# B&R Automation Studio project PLC code - cp (part 16)

#### AsignDataP5.st
```iecst
ACTION AsignDataP5:

	//Just writing the fixed configuration once per each 5s
	IF NOT (EDGEPOS(gPLC.xBlk_5s) OR gPLC.xFirst_Scan OR xChangedSimMachine) THEN
		RETURN;
	END_IF

	////////////////////////////////////////////////////////////
	/////GENERAL	GENERAL		GENERAL		GENERAL	////////////
	////////////////////////////////////////////////////////////

	gMachine.Pt.xControlledRemotely := FALSE;

	gMachine.Pt.CT.rMountedMediaLevelInBypassMode		:= 120.0;
	gMachine.Pt.CT.rMaxTicknessMedia		:= 120.0;
	gMachine.Pt.CT.rMinTicknessMedia		:= 2.0;
	gMachine.Pt.CT.iNumSAIInstalled			:= 2;

	gMachine.Pt.rMaxPrintHeadPos			:= 1668.0;
	gMachine.Pt.rMinPrintHeadPos			:= 10;
	gMachine.Pt.CT.rMinMarginPrinting		:= 1.0;

	gMachine.Pt.iMediaFilter 				:= 0;

	gMachine.Pt.PDSignalTpe 				:= PDCFG_SENSOR_AND_CARRIAGE;
	gMachine.Pt.xProtectPHWithStoppedMediaBended:= TRUE;
	gMachine.Pt.xProtectPHForBlowersRunning		:= FALSE;
	gMachine.Pt.Clean.xCleanBeltTopInstall 		:= FALSE;
	gMachine.Pt.xAllowLaboratory	 			:= TRUE;
	gMachine.Pt.xAllowJamRecovery	 			:= FALSE;
	gMachine.Pt.xJobNotReadyIsCritical	 		:= FALSE;
	gMachine.Pt.Clean.xCleanBeltForUv			:= FALSE;
	gMachine.Pt.CommsType						:= Type_ModbusTcp;

	gMachine.Pt.Hw.iWidth					:= 1440;
	gMachine.Pt.Hw.rMinPrintPosition		:= 2.0;
	gMachine.Pt.Hw.iMaxCuringLedBars		:= 0;
	gMachine.Pt.Hw.xDoubleLineAllowed		:= TRUE;
	gMachine.Pt.Hw.xSuctionModeAllowed		:= FALSE;

	gMachine.St.HwData.xIsPlatform5			:= TRUE;
	gMachine.St.HwData.xIsWater				:= gMachine.Pt.MachineModel=Type_P5_WTR;
	gMachine.St.HwData.xIsCubik				:= FALSE;

	//Belt
	gBelt.parameters.xRemoteAcceleration := FALSE;
	gBelt.parameters.xRemoteDeceleration := FALSE;
	gBelt.parameters.rAcceleration := 1050;
	gBelt.parameters.rDeceleration := 1050;
	gBelt.parameters.rMaxAcceleration := 1500.0;
	gBelt.parameters.rMaxDeceleration := 2500.0;

	//Here are configured blocks in function of the machine direction
	//When machine is block then we need use correction as block physical 2 because PD is at the same distance than Block 1, for that is change process in function of machine 2 Blcoks or machine 1 block
	gBlock[1].parameters.iMotorAxisIndex := 2;
	gBlock[1].parameters.iMappingBlock := 1;
	gBlock[1].parameters.iIclaAxisIndex := 1;
	gBlock[1].parameters.Hw.ValvesCommsType := COMMS_POWERLINK;

	/////////////////////////////////////////////////////
	// Temperature Modules Check
	////////////////////////////////////////////////////
	IF	NOT(gInks[1].parSw.Temp.xTankHeaterEnabled OR
		gInks[2].parSw.Temp.xTankHeaterEnabled OR
		gInks[3].parSw.Temp.xTankHeaterEnabled OR
		gInks[4].parSw.Temp.xTankHeaterEnabled) THEN

		gBlock[1].parameters.Inks.xTankHeatEnabled1 := FALSE;
	ELSE
		gBlock[1].parameters.Inks.xTankHeatEnabled1 := TRUE;
	END_IF

	IF	NOT(gInks[5].parSw.Temp.xTankHeaterEnabled OR
		gInks[6].parSw.Temp.xTankHeaterEnabled OR
		gInks[7].parSw.Temp.xTankHeaterEnabled OR
		gInks[8].parSw.Temp.xTankHeaterEnabled) THEN

		gBlock[1].parameters.Inks.xTankHeatEnabled2 := FALSE;
	ELSE
		gBlock[1].parameters.Inks.xTankHeatEnabled2 := TRUE;
	END_IF

	/////////////////////////////////////////////////////
	/////BELT	BELT	BELT	BELT	BELT	BELT/////
	/////////////////////////////////////////////////////

	////////////////////////////////////////////////////////////
	/////BLOCK	BLOCK	BLOCK	BLOCK	BLOCK	BLOCK///////////
	////////////////////////////////////////////////////////////
	FOR iIndexBlock:=1 TO gMachine.Pt.CT.iNumBlocks DO

		//Position parameters (mm)
		gBlock[iIndexBlock].parameters.Motor.rSafePosition				:= 356.0;//Max heigh
		gBlock[iIndexBlock].parameters.Motor.rMinSafePosition			:= 5.0;	 //Min heigh
		gBlock[iIndexBlock].parameters.Motor.rCapPosition				:= 344.0;//CAP
		gBlock[iIndexBlock].parameters.Motor.rSafePositionCleanCarrier	:= 329.0;//Carrier out Safe
		gBlock[iIndexBlock].parameters.Motor.rDripBarsPosition			:= 279.0;//Drip
		gBlock[iIndexBlock].parameters.Motor.rCleanPosition				:= 335.0;//Clean
		gBlock[iIndexBlock].parameters.Motor.rWaterSpurtPosition		:= 342.0;//Water Spurt
		gBlock[iIndexBlock].parameters.rPrePrintingPos					:= 75.0;  //PrePrinting Position

		gBlock[iIndexBlock].parameters.Motor.rAutoSpeedMoveDown	:=15.0;
		gBlock[iIndexBlock].parameters.Motor.rAutoSpeedMoveUp	:=30.0;
		gBlock[iIndexBlock].parameters.Motor.xFastSpeedAllowed	:= FALSE;

		gBlock[iIndexBlock].parameters.Motor.DriveUnit.TransmissionType := TRANS_SCREW_PITCH;
		gBlock[iIndexBlock].parameters.Motor.DriveUnit.ScrewPitch.PulsesPerTurn := GC_UNITS_BY_REV_DRIVE;
		gBlock[iIndexBlock].parameters.Motor.DriveUnit.ScrewPitch.GearBox := 7.25;
		gBlock[iIndexBlock].parameters.Motor.DriveUnit.ScrewPitch.Pitch := 5.0;

		gBlock[iIndexBlock].parameters.Motor.rReferencePosition		:= 15.5;

		//Current Parameters
		gBlock[iIndexBlock].parameters.Motor.uiMaxCurrentBarsUp			:= 3;
		gBlock[iIndexBlock].parameters.Motor.uiMaxCurrentBarsDown		:= 1;

		gBlock[iIndexBlock].parameters.Motor.VerticalDirection:= MOTOR_POSITIVE;

		gBlock[iIndexBlock].parameters.Motor.rAcceleration		:= 172.5;
		gBlock[iIndexBlock].parameters.Motor.rDeceleration		:= 172.5;

		gBlock[iIndexBlock].parameters.Icla.DriveUnit.TransmissionType:=TRANS_LINEAL_PERIMETER;
		gBlock[iIndexBlock].parameters.Icla.DriveUnit.LinealPerimeter.GearBox:=92;
		gBlock[iIndexBlock].parameters.Icla.DriveUnit.LinealPerimeter.Perimeter:=180;
		gBlock[iIndexBlock].parameters.Icla.DriveUnit.LinealPerimeter.PulsesPerTurn:=12;

		gBlock[iIndexBlock].parameters.Inks.iMaxMachinePrintBars	:= 8;
		gBlock[iIndexBlock].parameters.Inks.iMaxBlockPrintBars		:= 8;
		gBlock[iIndexBlock].parameters.Inks.iMaxPSUwattsForBars		:= 3000;

		gBlock[iIndexBlock].parameters.xCappingProcess := FALSE;

		gBlock[iIndexBlock].parameters.Hw.SafetySignals := SAFETY_ESTOP_CALCULATED;

		//[RGP] Due to issue SUSTPLATF-236
		gBlock[iIndexBlock].parameters.xMotorOffsetAllowed := FALSE;

		gBlock[iIndexBlock].parameters.iApplicationBars := 8;
	END_FOR

	///////////////////////////////////////////////////
	/////PHOTOCELLS		PHOTOCELLS		PHOTOCELLS/////
	///////////////////////////////////////////////////

	gPhotoCells.parameters.xInstall := TRUE;
	gMachine.parSw.Hw.xInstallnSensor := FALSE;
	gPhotoCells.parameters.xSensorsPosHybridBehaviour := FALSE;

	gPhotoCells.parameters.MotorType := STP_STEPPER;
	gPhotoCells.parameters.AlignmentProcess := STP_ALIGNMENT_NO_REQUIRED;

	gPhotoCells.parameters.Speed:=2.5;
	gPhotoCells.parameters.JogSpeed:=1;
	gPhotoCells.parameters.Acceleration:=5;

	gPhotoCells.parameters.DriveUnit.TransmissionType := TRANS_SCREW_PITCH;
	gPhotoCells.parameters.DriveUnit.ScrewPitch.PulsesPerTurn := GC_UNITS_BY_REV_DRIVE;
	gPhotoCells.parameters.DriveUnit.ScrewPitch.GearBox := 1;
	gPhotoCells.parameters.DriveUnit.ScrewPitch.Pitch := 2.5;

	IF gMachine.Pt.ConfigNameID = GC_CONFIG_SIMTEST_ID THEN
		// In Simulation
		gPhotoCells.parameters.IndexDriveMaster:=4;
		gPhotoCells.parameters.IndexDriveSecondary:=5;
	ELSE
		gPhotoCells.parameters.IndexDriveMaster:=3;
		gPhotoCells.parameters.IndexDriveSecondary:=4;
	END_IF

	gPhotoCells.parameters.iSensorQuantity := 3;
	gPhotoCells.parameters.iSensorToReference := 2;
	gPhotoCells.parameters.rOffsetPosition := 0.0;
	gPhotoCells.parameters.rSensorMechPositionByPass := 60.0;//110.0; //ALX -> ToReview
	gPhotoCells.parameters.Sensors[2].rDistanceRelativeToFirstSensor := 4;
	gPhotoCells.parameters.Sensors[3].rDistanceRelativeToFirstSensor := 8;
	gPhotoCells.parameters.xEnableMountedAlrByPass := TRUE;

	//Digital Inputs
	gPhotoCells.Inputs.Signals.pInput[1] := ADR(X20DIF371_003.DInput[13]);
	gPhotoCells.Inputs.Signals.pInput[2] := ADR(X20DIF371_003.DInput[14]);
	gPhotoCells.Inputs.Signals.pInput[3] := ADR(X20DIF371_003.DInput[15]);
	gPhotoCells.Inputs.Signals.xSafetyEnable := gMachine.In.xSafetyEnabled;

	stepperMotor ACCESS ADR (gAxis[gPhotoCells.parameters.IndexDriveMaster]);
	stepperMotor.Parameter.Direction:= MOTOR_NEGATIVE_AXIS;

	///////////////////////////////////////////////////
	/////DING		DING		DING		DING  /////
	///////////////////////////////////////////////////
	gDing.Parameters.xDingInstalled := FALSE;

	/////////////////////////////////////////////////////
	/////THICKNESS		THICKNESS		 THICKNESS///////
	/////////////////////////////////////////////////////

	gThicknessCtrl.parameters.iTotalBlocksLengh := 305;
	gThicknessCtrl.parameters.Belt.iDistanceEmptyBeltIni := 455; //The difference between Long and NotLong machine is 1350mm by side [700-135=615]

	gThicknessCtrl.parameters.xMarginForBendTile := TRUE;
	gThicknessCtrl.parameters.rSafetyMarginToHeight := 3.0;

	gThicknessCtrl.parameters.sections[1].xEnabled	:= TRUE;
	gThicknessCtrl.parameters.sections[1].iStart	:= 1;
	gThicknessCtrl.parameters.sections[1].iEnd		:= 305;

	gThicknessCtrl.parameters.Detection.ProductDetect.xLoadMedia := FALSE;
	gThicknessCtrl.parameters.Detection.ProductDetect.iSensorPosition := 25;
	gThicknessCtrl.parameters.Detection.Array.xLoadMedia := TRUE;
	gThicknessCtrl.parameters.Detection.Analog.iSensorPosition := 0;
	gThicknessCtrl.parameters.Detection.Analog.xLoadMedia := TRUE;
	gThicknessCtrl.parameters.Detection.Array.iSensorPosition := 0;

	/////////////////////////////////////////////////////
	/////   TRANSPORT_VACUUM  TRANSPORT_VACUUM   ////////
	/////////////////////////////////////////////////////
	gTransVacuum[1].Parameters.xInstalled := FALSE;
	gTransVacuum[2].Parameters.xInstalled := FALSE;

	/////////////////////////////////////////////////////
	/////   NON_CRASH    NON_CRASH    NON_CRASH  ////////
	/////////////////////////////////////////////////////
	gNonCrash[1].Parameters.xInstalled := FALSE;

	/////////////////////////////////////////////////////
	/////   PLC CARDS	PLC CARDS	PLC CARDS	 ////////
	/////////////////////////////////////////////////////
	IF gPlcCards[0].Type <> CARD_UNDEFINED THEN
		RETURN;
	END_IF

	//Force "ModuleOk" in cards without it
	X20CPUData.ModuleOk := TRUE;

	AsignCardsP5;

END_ACTION

ACTION AsignCardsP5:

	gPlcCards[0].Type := CARD_CPU0484;
	gPlcCards[0].pCard := ADR(X20CPUData);
	gPlcCards[0].RequiredForFunctions[0] := CARDREQUIRED_ALWAYS;
	gPlcCards[0].stCardName := 'X20CP0483_000';
	gPlcCards[0].Location := CardInPrinter;
	iIndexPlcCar := 1;

	//CARD 01 X20DIF371
	gPlcCards[iIndexPlcCar].Type := CARD_DI16;
	gPlcCards[iIndexPlcCar].pCard := ADR(X20DIF371_001);
	gPlcCards[iIndexPlcCar].RequiredForFunctions[0] := CARDREQUIRED_ALWAYS;
	gPlcCards[iIndexPlcCar].stCardName := 'X20DIF371-001';
	gPlcCards[iIndexPlcCar].Texts[1].Details := 'Machine Config-Bit 0';
	gPlcCards[iIndexPlcCar].Texts[2].Details := 'Machine Config-Bit 1';
	gPlcCards[iIndexPlcCar].Texts[3].Details := 'Machine Config-Bit 2';
	gPlcCards[iIndexPlcCar].Texts[4].Details := 'Machine Config-Bit 3';
	gPlcCards[iIndexPlcCar].Texts[5].Details := 'Machine Config-Bit 4';
	gPlcCards[iIndexPlcCar].Texts[6].Details := 'Machine Config-Bit 5';
	gPlcCards[iIndexPlcCar].Texts[7].Details := 'Start';
	gPlcCards[iIndexPlcCar].Texts[8].Details := 'Stop';
	gPlcCards[iIndexPlcCar].Texts[9].Details := 'Automatic';
	gPlcCards[iIndexPlcCar].Texts[10].Details := 'Zero';
	gPlcCards[iIndexPlcCar].Texts[11].Details := 'Manual';
	gPlcCards[iIndexPlcCar].Texts[12].Details := 'Validation to PLC';
	gPlcCards[iIndexPlcCar].Texts[13].Details := 'CB to PLC - Print Trigger L1';
	gPlcCards[iIndexPlcCar].Texts[14].Details := 'CB to PLC - Print Trigger L2';
	gPlcCards[iIndexPlcCar].Texts[15].Details := 'Spare';
	gPlcCards[iIndexPlcCar].Texts[16].Details := 'Spare';
	gPlcCards[iIndexPlcCar].Location := CardInPrinter;
	iIndexPlcCar := iIndexPlcCar + 1;

	//CARD 02 X20DIF371
	gPlcCards[iIndexPlcCar].Type := CARD_DI16;
	gPlcCards[iIndexPlcCar].pCard := ADR(X20DIF371_002);
	gPlcCards[iIndexPlcCar].RequiredForFunctions[0] := CARDREQUIRED_ALWAYS;
	gPlcCards[iIndexPlcCar].stCardName := 'X20DIF371-002';
	gPlcCards[iIndexPlcCar].Texts[1].Details := 'Bar A-48 VDC POWER OK';
	gPlcCards[iIndexPlcCar].Texts[2].Details := 'Bar B-48 VDC POWER OK';
	gPlcCards[iIndexPlcCar].Texts[3].Details := 'Bar C-48 VDC POWER OK';
	gPlcCards[iIndexPlcCar].Texts[4].Details := 'Bar D-48 VDC POWER OK';
	gPlcCards[iIndexPlcCar].Texts[5].Details := 'Bar E-48 VDC POWER OK';
	gPlcCards[iIndexPlcCar].Texts[6].Details := 'Bar F-48 VDC POWER OK';
	gPlcCards[iIndexPlcCar].Texts[7].Details := 'Bar G-48 VDC POWER OK';
	gPlcCards[iIndexPlcCar].Texts[8].Details := 'Bar H-48 VDC POWER OK';
	gPlcCards[iIndexPlcCar].Texts[9].Details := 'Bars heater - 48 VDC POWER OK';
	gPlcCards[iIndexPlcCar].Texts[10].Details := 'Transp driver-Diff contact alarm';
	gPlcCards[iIndexPlcCar].Texts[11].Details := 'Elev. driver-CB contact alarm';
	gPlcCards[iIndexPlcCar].Texts[12].Details := '48 VDC PSUs-Diff contact alarm';
	gPlcCards[iIndexPlcCar].Texts[13].Details := '24 VDC PSUs-IDS power alarm';
	gPlcCards[iIndexPlcCar].Texts[14].Details := 'Front light curtain-Alarm';
	gPlcCards[iIndexPlcCar].Texts[15].Details := 'Back Safety Switch-Alarm';
	gPlcCards[iIndexPlcCar].Texts[16].Details := 'Safety module status-Safety OK';
	gPlcCards[iIndexPlcCar].Location := CardInPrinter;
	iIndexPlcCar := iIndexPlcCar + 1;

	//CARD 03 X20DIF371
	gPlcCards[iIndexPlcCar].Type := CARD_DI16;
	gPlcCards[iIndexPlcCar].pCard := ADR(X20DIF371_003);
	gPlcCards[iIndexPlcCar].RequiredForFunctions[0] := CARDREQUIRED_ALWAYS;
	gPlcCards[iIndexPlcCar].stCardName := 'X20DIF371-003';
	gPlcCards[iIndexPlcCar].Texts[1].Details := 'UPS 1 - Failure UPS';
	gPlcCards[iIndexPlcCar].Texts[2].Details := 'UPS 1 - Utility Failure';
	gPlcCards[iIndexPlcCar].Texts[3].Details := 'UPS 1 - Low Battery';
	gPlcCards[iIndexPlcCar].Texts[4].Details := 'UPS 1 - Inverter Failure';
	gPlcCards[iIndexPlcCar].Texts[5].Details := 'UPS 2 - Failure UPS';
	gPlcCards[iIndexPlcCar].Texts[6].Details := 'UPS 2 - Utility Failure';
	gPlcCards[iIndexPlcCar].Texts[7].Details := 'UPS 2 - Low Battery';
	gPlcCards[iIndexPlcCar].Texts[8].Details := 'UPS 2 - Inverter Failure';
	gPlcCards[iIndexPlcCar].Texts[9].Details := 'Bars ref. sensor - ON signal';
	gPlcCards[iIndexPlcCar].Texts[10].Details := 'Spare';
	gPlcCards[iIndexPlcCar].Texts[11].Details := 'PD - Broken sensor alarm';
	gPlcCards[iIndexPlcCar].Texts[12].Details := 'DPT - Broken sensor alarm';
	gPlcCards[iIndexPlcCar].Texts[13].Details := '3L - Detected tile (Photocell 1)';
	gPlcCards[iIndexPlcCar].Texts[14].Details := '3L - Bent tile (Photocell 2)';
	gPlcCards[iIndexPlcCar].Texts[15].Details := '3L - Mounted tile (Photocell 3)';
	gPlcCards[iIndexPlcCar].Texts[16].Details := 'Spare';
	gPlcCards[iIndexPlcCar].Location := CardInPrinter;
	iIndexPlcCar := iIndexPlcCar + 1;

	//CARD 04 X20DIF371
	gPlcCards[iIndexPlcCar].Type := CARD_DI16;
	gPlcCards[iIndexPlcCar].pCard := ADR(X20DIF371_004);
	gPlcCards[iIndexPlcCar].RequiredForFunctions[0] := CARDREQUIRED_ALWAYS;
	gPlcCards[iIndexPlcCar].stCardName := 'X20DIF371-004';
	gPlcCards[iIndexPlcCar].Texts[1].Details := 'Bar A - Klixon';
	gPlcCards[iIndexPlcCar].Texts[2].Details := 'Bar B - Klixon';
	gPlcCards[iIndexPlcCar].Texts[3].Details := 'Bar C - Klixon';
	gPlcCards[iIndexPlcCar].Texts[4].Details := 'Bar D - Klixon';
	gPlcCards[iIndexPlcCar].Texts[5].Details := 'Bar E - Klixon';
	gPlcCards[iIndexPlcCar].Texts[6].Details := 'Bar F - Klixon';
	gPlcCards[iIndexPlcCar].Texts[7].Details := 'Bar G - Klixon';
	gPlcCards[iIndexPlcCar].Texts[8].Details := 'Bar H - Klixon';
	gPlcCards[iIndexPlcCar].Texts[9].Details := 'Tank A - Empty Level';
	gPlcCards[iIndexPlcCar].Texts[10].Details := 'Tank B - Empty Level';
	gPlcCards[iIndexPlcCar].Texts[11].Details := 'Tank C - Empty Level';
	gPlcCards[iIndexPlcCar].Texts[12].Details := 'Tank D - Empty Level';
	gPlcCards[iIndexPlcCar].Texts[13].Details := 'Tank E - Empty Level';
	gPlcCards[iIndexPlcCar].Texts[14].Details := 'Tank F - Empty Level';
	gPlcCards[iIndexPlcCar].Texts[15].Details := 'Tank G - Empty Level';
	gPlcCards[iIndexPlcCar].Texts[16].Details := 'Tank H - Empty Level';
	gPlcCards[iIndexPlcCar].Location := CardInPrinter;
	iIndexPlcCar := iIndexPlcCar + 1;

	//CARD 05 X20DIF371
	gPlcCards[iIndexPlcCar].Type := CARD_DI16;
	gPlcCards[iIndexPlcCar].pCard := ADR(X20DIF371_005);
	gPlcCards[iIndexPlcCar].RequiredForFunctions[0] := CARDREQUIRED_ALWAYS;
	gPlcCards[iIndexPlcCar].stCardName := 'X20DIF371-005';
	gPlcCards[iIndexPlcCar].Texts[1].Details := 'Tank A - Full Level';
	gPlcCards[iIndexPlcCar].Texts[2].Details := 'Tank B - Full Level';
	gPlcCards[iIndexPlcCar].Texts[3].Details := 'Tank C - Full Level';
	gPlcCards[iIndexPlcCar].Texts[4].Details := 'Tank D - Full Level';
	gPlcCards[iIndexPlcCar].Texts[5].Details := 'Tank E - Full Level';
	gPlcCards[iIndexPlcCar].Texts[6].Details := 'Tank F - Full Level';
	gPlcCards[iIndexPlcCar].Texts[7].Details := 'Tank G - Full Level';
	gPlcCards[iIndexPlcCar].Texts[8].Details := 'Tank H - Full Level';
	gPlcCards[iIndexPlcCar].Texts[9].Details := 'Tank A - Pressure Switch';
	gPlcCards[iIndexPlcCar].Texts[10].Details := 'Tank B - Pressure Switch';
	gPlcCards[iIndexPlcCar].Texts[11].Details := 'Tank C - Pressure Switch';
	gPlcCards[iIndexPlcCar].Texts[12].Details := 'Tank D - Pressure Switch';
	gPlcCards[iIndexPlcCar].Texts[13].Details := 'Tank E - Pressure Switch';
	gPlcCards[iIndexPlcCar].Texts[14].Details := 'Tank F - Pressure Switch';
	gPlcCards[iIndexPlcCar].Texts[15].Details := 'Tank G - Pressure Switch';
	gPlcCards[iIndexPlcCar].Texts[16].Details := 'Tank H - Pressure Switch';
	gPlcCards[iIndexPlcCar].Location := CardInPrinter;
	iIndexPlcCar := iIndexPlcCar + 1;

	//CARD 06 X20DIF371
	gPlcCards[iIndexPlcCar].Type := CARD_DI16;
	gPlcCards[iIndexPlcCar].pCard := ADR(X20DIF371_006);
	gPlcCards[iIndexPlcCar].RequiredForFunctions[0] := CARDREQUIRED_ALWAYS;
	gPlcCards[iIndexPlcCar].stCardName := 'X20DIF371-006';
	gPlcCards[iIndexPlcCar].Texts[1].Details := 'PBF - Bit 0';
	gPlcCards[iIndexPlcCar].Texts[2].Details := 'PBF - Bit 1';
	gPlcCards[iIndexPlcCar].Texts[3].Details := 'PBF - Bit 2';
	gPlcCards[iIndexPlcCar].Texts[4].Details := 'PBF - Bit 3';
	gPlcCards[iIndexPlcCar].Texts[5].Details := 'PBF - Bit 4';
	gPlcCards[iIndexPlcCar].Texts[6].Details := 'PBF - Bit 5';
	gPlcCards[iIndexPlcCar].Texts[7].Details := 'PBF - Bit 6';
	gPlcCards[iIndexPlcCar].Texts[8].Details := 'PBF - Bit 7';
	gPlcCards[iIndexPlcCar].Texts[9].Details := 'PBF - Strobe';
	gPlcCards[iIndexPlcCar].Texts[10].Details := 'Consent Line-Machine 1';
	gPlcCards[iIndexPlcCar].Texts[11].Details := 'Consent Line-Machine 2';
	gPlcCards[iIndexPlcCar].Texts[12].Details := 'PH External Cleaning';
	gPlcCards[iIndexPlcCar].Texts[13].Details := 'RESERVED';
	gPlcCards[iIndexPlcCar].Texts[14].Details := 'RESERVED';
	gPlcCards[iIndexPlcCar].Texts[15].Details := 'Spare';
	gPlcCards[iIndexPlcCar].Texts[16].Details := 'Spare';
	gPlcCards[iIndexPlcCar].Location := CardInPrinter;
	iIndexPlcCar := iIndexPlcCar + 1;

	//CARD 07 PS
	gPlcCards[iIndexPlcCar].Type := CARD_PS33;
	gPlcCards[iIndexPlcCar].pCard := ADR(X20PS3300_007);
	gPlcCards[iIndexPlcCar].RequiredForFunctions[0] := CARDREQUIRED_ALWAYS;
	gPlcCards[iIndexPlcCar].stCardName := 'X20PS3300-007';
	gPlcCards[iIndexPlcCar].Location := CardInPrinter;
	iIndexPlcCar := iIndexPlcCar + 1;

	//CARD 8 X20DI9372
	gPlcCards[iIndexPlcCar].Type := CARD_DI16;
	gPlcCards[iIndexPlcCar].pCard := ADR(X20DI9372_008);
	gPlcCards[iIndexPlcCar].RequiredForFunctions[0] := CARDREQUIRED_ALWAYS;
	gPlcCards[iIndexPlcCar].stCardName := 'X20DI9372_008';
	gPlcCards[iIndexPlcCar].Texts[1].Details :='48VDC PSU 1 (PH) -48 V OK';
	gPlcCards[iIndexPlcCar].Texts[2].Details :='48VDC PSU 2 (PH) -48 V OK';
	gPlcCards[iIndexPlcCar].Texts[3].Details :='48VDC PSU 3 (PH) -48 V OK';
	gPlcCards[iIndexPlcCar].Texts[4].Details :='48VDC PSU 4 (PH) -48 V OK';
	gPlcCards[iIndexPlcCar].Texts[5].Details :='48VDC PSU 5 (PH) -48 V OK';
	gPlcCards[iIndexPlcCar].Texts[6].Details :='48VDC PSU 6 (PH) -48 V OK';
	gPlcCards[iIndexPlcCar].Texts[7].Details :='48VDC PSU 7 (Heat) -48 V OK';
	gPlcCards[iIndexPlcCar].Texts[8].Details :='48VDC PSU 8 (Heat) -48 V OK';
	gPlcCards[iIndexPlcCar].Texts[9].Details :='48VDC PSU 9 (Heat) -48 V OK';
	gPlcCards[iIndexPlcCar].Texts[10].Details :='Spare';
	gPlcCards[iIndexPlcCar].Texts[11].Details :='Spare';
	gPlcCards[iIndexPlcCar].Texts[12].Details :='Spare';
	gPlcCards[iIndexPlcCar].Location := CardInPrinter;
	iIndexPlcCar := iIndexPlcCar + 1;

	//CARD 9 X20DOF322
	gPlcCards[iIndexPlcCar].Type := CARD_DO16;
	gPlcCards[iIndexPlcCar].pCard := ADR(X20DOF322_009);
	gPlcCards[iIndexPlcCar].RequiredForFunctions[0] := CARDREQUIRED_ALWAYS;
	gPlcCards[iIndexPlcCar].stCardName := 'X20DOF322_009';
	gPlcCards[iIndexPlcCar].Texts[1].Details :='PLC to CB-Simulation PD1';
	gPlcCards[iIndexPlcCar].Texts[2].Details :='PLC to CB-Simulation PD2';
	gPlcCards[iIndexPlcCar].Texts[3].Details :='DTP Enable';
	gPlcCards[iIndexPlcCar].Texts[4].Details :='Reset Carriage Board 1&2';
	gPlcCards[iIndexPlcCar].Texts[5].Details :='Reset Router';
	gPlcCards[iIndexPlcCar].Texts[6].Details :='Spare';
	gPlcCards[iIndexPlcCar].Texts[7].Details :='Zero mode - Air supply off';
	gPlcCards[iIndexPlcCar].Texts[8].Details :='Start Green Light ON';
	gPlcCards[iIndexPlcCar].Texts[9].Details :='Reset blue light ON';
	gPlcCards[iIndexPlcCar].Texts[10].Details :='Buzzer';
	gPlcCards[iIndexPlcCar].Texts[11].Details :='Status PLC-Run';
	gPlcCards[iIndexPlcCar].Texts[12].Details :='Spare';
	gPlcCards[iIndexPlcCar].Texts[13].Details :='Spare';
	gPlcCards[iIndexPlcCar].Texts[14].Details :='Spare';
	gPlcCards[iIndexPlcCar].Texts[15].Details :='Spare';
	gPlcCards[iIndexPlcCar].Texts[16].Details :='Spare';
	gPlcCards[iIndexPlcCar].Location := CardInPrinter;
	iIndexPlcCar := iIndexPlcCar + 1;

	//CARD 10 X20DOF322
	gPlcCards[iIndexPlcCar].Type := CARD_DO16;
	gPlcCards[iIndexPlcCar].pCard := ADR(X20DOF322_010);
	gPlcCards[iIndexPlcCar].RequiredForFunctions[0] := CARDREQUIRED_ALWAYS;
	gPlcCards[iIndexPlcCar].stCardName := 'X20DOF322_010';
	gPlcCards[iIndexPlcCar].Texts[1].Details :='BarA -PH power ON';
	gPlcCards[iIndexPlcCar].Texts[2].Details :='BarB -PH power ON';
	gPlcCards[iIndexPlcCar].Texts[3].Details :='BarC -PH power ON';
	gPlcCards[iIndexPlcCar].Texts[4].Details :='BarD -PH power ON';
	gPlcCards[iIndexPlcCar].Texts[5].Details :='BarE -PH power ON';
	gPlcCards[iIndexPlcCar].Texts[6].Details :='BarF -PH power ON';
	gPlcCards[iIndexPlcCar].Texts[7].Details :='BarG -PH power ON';
	gPlcCards[iIndexPlcCar].Texts[8].Details :='BarH -PH power ON';
	gPlcCards[iIndexPlcCar].Texts[9].Details :='BarA -Heating ON';
	gPlcCards[iIndexPlcCar].Texts[10].Details :='BarB -Heating ON';
	gPlcCards[iIndexPlcCar].Texts[11].Details :='BarC -Heating ON';
	gPlcCards[iIndexPlcCar].Texts[12].Details :='BarD -Heating ON';
	gPlcCards[iIndexPlcCar].Texts[13].Details :='BarE -Heating ON';
	gPlcCards[iIndexPlcCar].Texts[14].Details :='BarF -Heating ON';
	gPlcCards[iIndexPlcCar].Texts[15].Details :='BarG -Heating ON';
	gPlcCards[iIndexPlcCar].Texts[16].Details :='BarH -Heating ON';
	gPlcCards[iIndexPlcCar].Location := CardInPrinter;
	iIndexPlcCar := iIndexPlcCar + 1;

	//CARD 11 X20DOF322
	gPlcCards[iIndexPlcCar].Type := CARD_DO16;
	gPlcCards[iIndexPlcCar].pCard := ADR(X20DOF322_011);
	gPlcCards[iIndexPlcCar].RequiredForFunctions[0] := CARDREQUIRED_ALWAYS;
	gPlcCards[iIndexPlcCar].stCardName := 'X20DOF322_011';
	gPlcCards[iIndexPlcCar].Texts[1].Details :='BarA-Rev.Flow Solen.1-4';
	gPlcCards[iIndexPlcCar].Texts[2].Details :='BarB-Rev.Flow Solen.1-4';
	gPlcCards[iIndexPlcCar].Texts[3].Details :='BarA-Rev.Flow Solen.2-3';
	gPlcCards[iIndexPlcCar].Texts[4].Details :='BarB-Rev.Flow Solen.2-3';
	gPlcCards[iIndexPlcCar].Texts[5].Details :='BarC-Rev.Flow Solen.1-4';
	gPlcCards[iIndexPlcCar].Texts[6].Details :='BarD-Rev.Flow Solen.1-4';
	gPlcCards[iIndexPlcCar].Texts[7].Details :='BarC-Rev.Flow Solen.2-3';
	gPlcCards[iIndexPlcCar].Texts[8].Details :='BarD-Rev.Flow Solen.2-3';
	gPlcCards[iIndexPlcCar].Texts[9].Details :='BarE-Rev.Flow Solen.1-4';
	gPlcCards[iIndexPlcCar].Texts[10].Details :='BarF-Rev.Flow Solen.1-4';
	gPlcCards[iIndexPlcCar].Texts[11].Details :='BarE-Rev.Flow Solen.2-3';
	gPlcCards[iIndexPlcCar].Texts[12].Details :='BarF-Rev.Flow Solen.2-3';
	gPlcCards[iIndexPlcCar].Texts[13].Details :='BarG-Rev.Flow Solen.1-4';
	gPlcCards[iIndexPlcCar].Texts[14].Details :='BarH-Rev.Flow Solen.1-4';
	gPlcCards[iIndexPlcCar].Texts[15].Details :='BarG-Rev.Flow Solen.2-3';
	gPlcCards[iIndexPlcCar].Texts[16].Details :='BarH-Rev.Flow Solen.2-3';
	gPlcCards[iIndexPlcCar].Location := CardInPrinter;
	iIndexPlcCar := iIndexPlcCar + 1;

	//CARD 12 X20DOF322
	gPlcCards[iIndexPlcCar].Type := CARD_DO16;
	gPlcCards[iIndexPlcCar].pCard := ADR(X20DOF322_012);
	gPlcCards[iIndexPlcCar].RequiredForFunctions[0] := CARDREQUIRED_ALWAYS;
	gPlcCards[iIndexPlcCar].stCardName := 'X20DOF322_012';
	gPlcCards[iIndexPlcCar].Texts[1].Details :='BarA-Minifold tank EV';
	gPlcCards[iIndexPlcCar].Texts[2].Details :='BarB-Minifold tank EV';
	gPlcCards[iIndexPlcCar].Texts[3].Details :='BarC-Minifold tank EV';
	gPlcCards[iIndexPlcCar].Texts[4].Details :='BarD-Minifold tank EV';
	gPlcCards[iIndexPlcCar].Texts[5].Details :='BarE-Minifold tank EV';
	gPlcCards[iIndexPlcCar].Texts[6].Details :='BarF-Minifold tank EV';
	gPlcCards[iIndexPlcCar].Texts[7].Details :='BarG-Minifold tank EV';
	gPlcCards[iIndexPlcCar].Texts[8].Details :='BarH-Minifold tank EV';
	gPlcCards[iIndexPlcCar].Texts[9].Details :='BarA-Preheat power ON';
	gPlcCards[iIndexPlcCar].Texts[10].Details :='BarB-Preheat power ON';
	gPlcCards[iIndexPlcCar].Texts[11].Details :='BarC-Preheat power ON';
	gPlcCards[iIndexPlcCar].Texts[12].Details :='BarD-Preheat power ON';
	gPlcCards[iIndexPlcCar].Texts[13].Details :='BarE-Preheat power ON';
	gPlcCards[iIndexPlcCar].Texts[14].Details :='BarF-Preheat power ON';
	gPlcCards[iIndexPlcCar].Texts[15].Details :='BarG-Preheat power ON';
	gPlcCards[iIndexPlcCar].Texts[16].Details :='BarH-Preheat power ON';
	gPlcCards[iIndexPlcCar].Location := CardInPrinter;
	iIndexPlcCar := iIndexPlcCar + 1;

	//CARD 13 X20DOF322
	gPlcCards[iIndexPlcCar].Type := CARD_DO16;
	gPlcCards[iIndexPlcCar].pCard := ADR(X20DOF322_013);
	gPlcCards[iIndexPlcCar].RequiredForFunctions[0] := CARDREQUIRED_ALWAYS;
	gPlcCards[iIndexPlcCar].stCardName := 'X20DOF322_013';
	gPlcCards[iIndexPlcCar].Texts[1].Details :='Consent Machine-Line1';
	gPlcCards[iIndexPlcCar].Texts[2].Details :='Consent Machine-Line2';
	gPlcCards[iIndexPlcCar].Texts[3].Details :='Compenser Line 1';
	gPlcCards[iIndexPlcCar].Texts[4].Details :='Compenser Line 2';
	gPlcCards[iIndexPlcCar].Texts[5].Details :='Warning Machine (Yellow)';
	gPlcCards[iIndexPlcCar].Texts[6].Details :='Emergency Machine (Red)';
	gPlcCards[iIndexPlcCar].Texts[7].Details :='Line 1 - Ready Clean Up';
	gPlcCards[iIndexPlcCar].Texts[8].Details :='Line 2 - Ready Clean Up';
	gPlcCards[iIndexPlcCar].Texts[9].Details :='Suction Tutbine';
	gPlcCards[iIndexPlcCar].Texts[10].Details :='Jam detection - Test sensors 1&5';
	gPlcCards[iIndexPlcCar].Texts[11].Details :='Jam detection - Test sensors 2&6';
	gPlcCards[iIndexPlcCar].Texts[12].Details :='Jam detection - Test sensors 3&7';
	gPlcCards[iIndexPlcCar].Texts[13].Details :='Jam detection - Test sensors 4&8';
	gPlcCards[iIndexPlcCar].Texts[14].Details :='Spare';
	gPlcCards[iIndexPlcCar].Texts[15].Details :='Sapre';
	gPlcCards[iIndexPlcCar].Texts[16].Details :='Spare';
	gPlcCards[iIndexPlcCar].Location := CardInPrinter;
	iIndexPlcCar := iIndexPlcCar + 1;

	//CARD 14 PS
	gPlcCards[iIndexPlcCar].Type := CARD_PS33;
	gPlcCards[iIndexPlcCar].pCard := ADR(X20PS3300_014);
	gPlcCards[iIndexPlcCar].RequiredForFunctions[0] := CARDREQUIRED_ALWAYS;
	gPlcCards[iIndexPlcCar].stCardName := 'X20PS3300-014';
	gPlcCards[iIndexPlcCar].Location := CardInPrinter;
	iIndexPlcCar := iIndexPlcCar + 1;

	//CARD 15 X20AI8321
	gPlcCards[iIndexPlcCar].Type := CARD_AI8;
	gPlcCards[iIndexPlcCar].pCard := ADR(X20AI8321_015);
	gPlcCards[iIndexPlcCar].RequiredForFunctions[0] := CARDREQUIRED_ALWAYS;
	gPlcCards[iIndexPlcCar].stCardName := 'X20AI8321_015';
	gPlcCards[iIndexPlcCar].Texts[1].Details :='BarA-Pos. Manif. Press. Sensor';
	gPlcCards[iIndexPlcCar].Texts[2].Details :='BarA-Neg. Manif. Press. Sensor';
	gPlcCards[iIndexPlcCar].Texts[3].Details :='BarB-Pos. Manif. Press. Sensor';
	gPlcCards[iIndexPlcCar].Texts[4].Details :='BarB-Neg. Manif. Press. Sensor';
	gPlcCards[iIndexPlcCar].Texts[5].Details :='BarC-Pos. Manif. Press. Sensor';
	gPlcCards[iIndexPlcCar].Texts[6].Details :='BarC-Neg. Manif. Press. Sensor';
	gPlcCards[iIndexPlcCar].Texts[7].Details :='BarD-Pos. Manif. Press. Sensor';
	gPlcCards[iIndexPlcCar].Texts[8].Details :='BarD-Neg. Manif. Press. Sensor';
	gPlcCards[iIndexPlcCar].Location := CardInPrinter;
	iIndexPlcCar := iIndexPlcCar + 1;

	//CARD 16 X20AI8321
	gPlcCards[iIndexPlcCar].Type := CARD_AI8;
	gPlcCards[iIndexPlcCar].pCard := ADR(X20AI8321_016);
	gPlcCards[iIndexPlcCar].RequiredForFunctions[0] := CARDREQUIRED_ALWAYS;
	gPlcCards[iIndexPlcCar].stCardName := 'X20AI8321_016';
	gPlcCards[iIndexPlcCar].Texts[1].Details :='BarE-Pos. Manif. Press. Sensor';
	gPlcCards[iIndexPlcCar].Texts[2].Details :='BarE-Neg. Manif. Press. Sensor';
	gPlcCards[iIndexPlcCar].Texts[3].Details :='BarF-Pos. Manif. Press. Sensor';
	gPlcCards[iIndexPlcCar].Texts[4].Details :='BarF-Neg. Manif. Press. Sensor';
	gPlcCards[iIndexPlcCar].Texts[5].Details :='BarG-Pos. Manif. Press. Sensor';
	gPlcCards[iIndexPlcCar].Texts[6].Details :='BarG-Neg. Manif. Press. Sensor';
	gPlcCards[iIndexPlcCar].Texts[7].Details :='BarH-Pos. Manif. Press. Sensor';
	gPlcCards[iIndexPlcCar].Texts[8].Details :='BarH-Neg. Manif. Press. Sensor';
	gPlcCards[iIndexPlcCar].Location := CardInPrinter;
	iIndexPlcCar := iIndexPlcCar + 1;

	//CARD 17 X20AO4622
	gPlcCards[iIndexPlcCar].Type := CARD_AO4;
	gPlcCards[iIndexPlcCar].pCard := ADR(X20AO4622_017);
	gPlcCards[iIndexPlcCar].RequiredForFunctions[0] := CARDREQUIRED_ALWAYS;
	gPlcCards[iIndexPlcCar].stCardName := 'X20AO4622_017';
	gPlcCards[iIndexPlcCar].Texts[1].Details :='Tank A - Pump Negative';
	gPlcCards[iIndexPlcCar].Texts[2].Details :='Tank B - Pump Negative';
	gPlcCards[iIndexPlcCar].Texts[3].Details :='Tank A - Pump Positive';
	gPlcCards[iIndexPlcCar].Texts[4].Details :='Tank B - Pump Positive';
	gPlcCards[iIndexPlcCar].Location := CardInPrinter;
	iIndexPlcCar := iIndexPlcCar + 1;

	//CARD 18 X20AO4622
	gPlcCards[iIndexPlcCar].Type := CARD_AO4;
	gPlcCards[iIndexPlcCar].pCard := ADR(X20AO4622_018);
	gPlcCards[iIndexPlcCar].RequiredForFunctions[0] := CARDREQUIRED_ALWAYS;
	gPlcCards[iIndexPlcCar].stCardName := 'X20AO4622_018';
	gPlcCards[iIndexPlcCar].Texts[1].Details :='Tank C - Pump Negative';
	gPlcCards[iIndexPlcCar].Texts[2].Details :='Tank D - Pump Negative';
	gPlcCards[iIndexPlcCar].Texts[3].Details :='Tank C - Pump Positive';
	gPlcCards[iIndexPlcCar].Texts[4].Details :='Tank D - Pump Positive';
	gPlcCards[iIndexPlcCar].Location := CardInPrinter;
	iIndexPlcCar := iIndexPlcCar + 1;

	//CARD 19 X20AO4622
	gPlcCards[iIndexPlcCar].Type := CARD_AO4;
	gPlcCards[iIndexPlcCar].pCard := ADR(X20AO4622_019);
	gPlcCards[iIndexPlcCar].RequiredForFunctions[0] := CARDREQUIRED_ALWAYS;
	gPlcCards[iIndexPlcCar].stCardName := 'X20AO4622_019';
	gPlcCards[iIndexPlcCar].Texts[1].Details :='Tank E - Pump Negative';
	gPlcCards[iIndexPlcCar].Texts[2].Details :='Tank F - Pump Negative';
	gPlcCards[iIndexPlcCar].Texts[3].Details :='Tank E - Pump Positive';
	gPlcCards[iIndexPlcCar].Texts[4].Details :='Tank F - Pump Positive';
	gPlcCards[iIndexPlcCar].Location := CardInPrinter;
	iIndexPlcCar := iIndexPlcCar + 1;

	//CARD 20 X20AO4622
	gPlcCards[iIndexPlcCar].Type := CARD_AO4;
	gPlcCards[iIndexPlcCar].pCard := ADR(X20AO4622_020);
	gPlcCards[iIndexPlcCar].RequiredForFunctions[0] := CARDREQUIRED_ALWAYS;
	gPlcCards[iIndexPlcCar].stCardName := 'X20AO4622_020';
	gPlcCards[iIndexPlcCar].Texts[1].Details :='Tank G - Pump Negative';
	gPlcCards[iIndexPlcCar].Texts[2].Details :='Tank H - Pump Negative';
	gPlcCards[iIndexPlcCar].Texts[3].Details :='Tank G - Pump Positive';
	gPlcCards[iIndexPlcCar].Texts[4].Details :='Tank H - Pump Positive';
	gPlcCards[iIndexPlcCar].Location := CardInPrinter;
	iIndexPlcCar := iIndexPlcCar + 1;

	//CARD 21 PS
	gPlcCards[iIndexPlcCar].Type := CARD_PS33;
	gPlcCards[iIndexPlcCar].pCard := ADR(X20PS3300_021);
	gPlcCards[iIndexPlcCar].RequiredForFunctions[0] := CARDREQUIRED_ALWAYS;
	gPlcCards[iIndexPlcCar].stCardName := 'X20PS3300-021';
	gPlcCards[iIndexPlcCar].Location := CardInPrinter;
	iIndexPlcCar := iIndexPlcCar + 1;

	//CARD 22 X20AT4222
	gPlcCards[iIndexPlcCar].Type := CARD_AT4;
	gPlcCards[iIndexPlcCar].pCard := ADR(X20AT4222_022);
	gPlcCards[iIndexPlcCar].RequiredForFunctions[0] := CARDREQUIRED_ALWAYS;
	gPlcCards[iIndexPlcCar].stCardName := 'X20AT4222_022';
	gPlcCards[iIndexPlcCar].Texts[1].Details :='BarA - Temp. Probe (Manifold)';
	gPlcCards[iIndexPlcCar].Texts[2].Details :='BarB - Temp. Probe (Manifold)';
	gPlcCards[iIndexPlcCar].Texts[3].Details :='BarC - Temp. Probe (Manifold)';
	gPlcCards[iIndexPlcCar].Texts[4].Details :='BarD - Temp. Probe (Manifold)';
	gPlcCards[iIndexPlcCar].Location := CardInPrinter;
	iIndexPlcCar := iIndexPlcCar + 1;

	//CARD 23 X20AT4222
	gPlcCards[iIndexPlcCar].Type := CARD_AT4;
	gPlcCards[iIndexPlcCar].pCard := ADR(X20AT4222_023);
	gPlcCards[iIndexPlcCar].RequiredForFunctions[0] := CARDREQUIRED_ALWAYS;
	gPlcCards[iIndexPlcCar].stCardName := 'X20AT4222_023';
	gPlcCards[iIndexPlcCar].Texts[1].Details :='BarE - Temp. Probe (Manifold)';
	gPlcCards[iIndexPlcCar].Texts[2].Details :='BarF - Temp. Probe (Manifold)';
	gPlcCards[iIndexPlcCar].Texts[3].Details :='BarG - Temp. Probe (Manifold)';
	gPlcCards[iIndexPlcCar].Texts[4].Details :='BarH - Temp. Probe (Manifold)';
	gPlcCards[iIndexPlcCar].Location := CardInPrinter;
	iIndexPlcCar := iIndexPlcCar + 1;

	//CARD 24 Stepper Driver
	gPlcCards[iIndexPlcCar].Type := CARD_SM;
	gPlcCards[iIndexPlcCar].pCard := ADR(X20SM1436_111);
	gPlcCards[iIndexPlcCar].RequiredForFunctions[0] := CARDREQUIRED_SENSOR_THICK;
	gPlcCards[iIndexPlcCar].stCardName := 'X20SM1436_111';
	gPlcCards[iIndexPlcCar].Location := CardInPrinter;
	iIndexPlcCar := iIndexPlcCar + 1;

	//CARD 25 Stepper Driver
	gPlcCards[iIndexPlcCar].Type := CARD_SM;
	gPlcCards[iIndexPlcCar].pCard := ADR(X20SM1436_112);
	gPlcCards[iIndexPlcCar].RequiredForFunctions[0] := CARDREQUIRED_SENSOR_THICK;
	gPlcCards[iIndexPlcCar].stCardName := 'X20SM1436_112';
	gPlcCards[iIndexPlcCar].Location := CardInPrinter;
	iIndexPlcCar := iIndexPlcCar + 1;

	//CARD 26 X20AT4222
	IF X20AT4222_120.ModuleOk THEN
		gPlcCards[iIndexPlcCar].Type := CARD_AT4;
		gPlcCards[iIndexPlcCar].pCard := ADR(X20AT4222_120);
		gPlcCards[iIndexPlcCar].RequiredForFunctions[0] := CARDREQUIRED_ALWAYS;
		gPlcCards[iIndexPlcCar].stCardName := 'X20AT4222_120';
		gPlcCards[iIndexPlcCar].Texts[1].Details :='TankA - Preheat. Temp. Probe';
		gPlcCards[iIndexPlcCar].Texts[2].Details :='TankB - Preheat. Temp. Probe';
		gPlcCards[iIndexPlcCar].Texts[3].Details :='TankC - Preheat. Temp. Probe';
		gPlcCards[iIndexPlcCar].Texts[4].Details :='TankD - Preheat. Temp. Probe';
		gPlcCards[iIndexPlcCar].Location := CardInPrinter;
		iIndexPlcCar := iIndexPlcCar + 1;
	END_IF

	//CARD 27 X20AT4222
	IF X20AT4222_121.ModuleOk THEN
		gPlcCards[iIndexPlcCar].Type := CARD_AT4;
		gPlcCards[iIndexPlcCar].pCard := ADR(X20AT4222_121);
		gPlcCards[iIndexPlcCar].RequiredForFunctions[0] := CARDREQUIRED_ALWAYS;
		gPlcCards[iIndexPlcCar].stCardName := 'X20AT4222_121';
		gPlcCards[iIndexPlcCar].Texts[1].Details :='TankE - Preheat. Temp. Probe';
		gPlcCards[iIndexPlcCar].Texts[2].Details :='TankF - Preheat. Temp. Probe';
		gPlcCards[iIndexPlcCar].Texts[3].Details :='TankG - Preheat. Temp. Probe';
		gPlcCards[iIndexPlcCar].Texts[4].Details :='TankH - Preheat. Temp. Probe';
		gPlcCards[iIndexPlcCar].Location := CardInPrinter;
		iIndexPlcCar := iIndexPlcCar + 1;
	END_IF

	//END CARDS

	gPlcCards[iIndexPlcCar].Type := CARD_UNDEFINED;

END_ACTION
```

#### AsignDataPlcDiagnosis.st
```iecst
ACTION AsignDataPlcDiagnosis:

	CASE gPlcDiagMC_Pt.ConfigNameID OF

		GC_CONFIG_2BK12BAR_ID:
			AsignDataP4;

		GC_CONFIG_1BK2BAR_ID:
			AsignDataShld;

		GC_CONFIG_BM_1BK8BAR_ID:
			CASE gPlcDiagMC_Pt.MachineModel OF
				Type_S1400,
				Type_P5_OIL,
				Type_P5_WTR:
					AsignDataP5;
					Type_S1400_VAC_PWRLNK,
				Type_S1400_VAC_CAN:
					AsignDataS1400;
			END_CASE

		GC_CONFIG_1BK8BAR_NOZ2_ID:
			CASE gPlcDiagMC_Pt.MachineModel OF
				Type_NOZ_2_AQ,
				Type_NOZ_2_UV,
				Type_NOZ_2_UV_White:
					AsignDataNozomi2;
			END_CASE

		GC_CONFIG_1BK8BAR_NOZ2_AQ_ID:
			CASE gPlcDiagMC_Pt.MachineModel OF
				Type_NOZ_2_AQ:
					AsignDataNozomi2;
			END_CASE

		GC_CONFIG_1BK7BAR_CUBE_ID:
			CASE gPlcDiagMC_Pt.MachineModel OF
				Type_CUBE,
				Type_CUBE_INSPECTION,
				Type_CUBE_GULLIVER,
				Type_CUBE_GULLIVER_INSPECTION:
					AsignDataCube;
			END_CASE

		GC_CONFIG_1BK10BAR_MECANO_ID:
			CASE gPlcDiagMC_Pt.MachineModel OF
				Type_MECANO_UV_WHITE,
				Type_MECANO_UV_OPV,
				Type_MECANO_UV_WHITE_OPV:
					AssignDataMecano;
			END_CASE

	END_CASE

END_ACTION
```

#### AsignDataShld.st
```iecst
ACTION AsignDataShld:

	//Just writing the fixed configuration once per each 5s
	IF NOT (EDGEPOS(gPLC.xBlk_5s) OR gPLC.xFirst_Scan OR xChangedSimMachine) THEN
		RETURN;
	END_IF

	////////////////////////////////////////////////////////////
	/////GENERAL	GENERAL		GENERAL		GENERAL	////////////
	////////////////////////////////////////////////////////////

	gMachine.Pt.xControlledRemotely := FALSE;

	gMachine.Pt.CT.rMountedMediaLevelInBypassMode		:= 60.0;
	gMachine.Pt.CT.rMaxTicknessMedia		:= 60.0;
	gMachine.Pt.CT.rMinTicknessMedia		:= 2.0;
	gMachine.Pt.CT.iNumSAIInstalled			:= 1;

	gMachine.Pt.rMaxPrintHeadPos			:= 1623.0;
	gMachine.Pt.rMinPrintHeadPos			:= 10;
	gMachine.Pt.CT.rMinMarginPrinting		:= 1.0;

	gMachine.Pt.iMediaFilter 				:= 0;

	gMachine.Pt.PDSignalTpe 						:= PDCFG_SENSOR_AND_CARRIAGE;
	gMachine.Pt.xProtectPHWithStoppedMediaBended	:= TRUE;
	gMachine.Pt.xProtectPHForBlowersRunning			:= FALSE;
	gMachine.Pt.Clean.xCleanBeltTopInstall 				:= FALSE;
	gMachine.Pt.xAllowLaboratory	 				:= TRUE;
	gMachine.Pt.xAllowJamRecovery	 				:= FALSE;
	gMachine.Pt.xJobNotReadyIsCritical	 			:= FALSE;
	gMachine.Pt.Clean.xCleanBeltForUv						:= FALSE;
	gMachine.Pt.CommsType							:= Type_ModbusTcp;

	gMachine.Pt.Hw.iWidth					:= 1440;
	gMachine.Pt.Hw.rMinPrintPosition		:= 2.0;
	gMachine.Pt.Hw.iMaxCuringLedBars		:= 0;
	gMachine.Pt.Hw.xDoubleLineAllowed		:= TRUE;
	gMachine.Pt.Hw.xSuctionModeAllowed		:= FALSE;

	gMachine.St.HwData.xIsPlatform5			:= TRUE;
	gMachine.St.HwData.xIsWater				:= TRUE;
	gMachine.St.HwData.xIsCubik				:= FALSE;

	//Belt
	gBelt.parameters.xRemoteAcceleration := FALSE;
	gBelt.parameters.xRemoteDeceleration := FALSE;
	gBelt.parameters.rAcceleration := 1050;
	gBelt.parameters.rDeceleration := 1050;
	gBelt.parameters.rMaxAcceleration := 1500.0;
	gBelt.parameters.rMaxDeceleration := 2500.0;

	//Here are configured blocks in function of the machine direction
	//When machine is block then we need use correction as block physical 2 because PD is at the same distance than Block 1, for that is change process in function of machine 2 Blcoks or machine 1 block
	gBlock[1].parameters.iMotorAxisIndex := 2;
	gBlock[1].parameters.iMappingBlock := 1;
	gBlock[1].parameters.iIclaAxisIndex := 1;
	gBlock[1].parameters.Hw.ValvesCommsType := COMMS_CANOPEN;
	gBlock[1].parameters.Hw.ValvesNode := 6;

	////////////////////////////////////////////////////////////
	/////BLOCK	BLOCK	BLOCK	BLOCK	BLOCK	BLOCK///////////
	////////////////////////////////////////////////////////////
	FOR iIndexBlock:=1 TO gMachine.Pt.CT.iNumBlocks DO

		//Position parameters (mm)
		gBlock[iIndexBlock].parameters.Motor.rSafePosition				:= 287.0;//3330;//Max heigh
		gBlock[iIndexBlock].parameters.Motor.rMinSafePosition			:= 5.0;	 //Min heigh
		gBlock[iIndexBlock].parameters.Motor.rCapPosition				:= 282.0;//3280;//CAP
		gBlock[iIndexBlock].parameters.Motor.rSafePositionCleanCarrier	:= 267.0;//Carrier out Safe
		gBlock[iIndexBlock].parameters.Motor.rDripBarsPosition			:= 218.0;//Drip
		gBlock[iIndexBlock].parameters.Motor.rCleanPosition				:= 273.0;//Clean
		gBlock[iIndexBlock].parameters.Motor.rWaterSpurtPosition		:= 281.0;//Water Spurt
		gBlock[iIndexBlock].parameters.rPrePrintingPos					:= 75.0;  //PrePrinting Position

		gBlock[iIndexBlock].parameters.Motor.rAutoSpeedMoveDown	:=30.0;
		gBlock[iIndexBlock].parameters.Motor.rAutoSpeedMoveUp	:=30.0;
		gBlock[iIndexBlock].parameters.Motor.xFastSpeedAllowed	:= FALSE;

		gBlock[iIndexBlock].parameters.Motor.DriveUnit.TransmissionType := TRANS_SCREW_PITCH;
		gBlock[iIndexBlock].parameters.Motor.DriveUnit.ScrewPitch.PulsesPerTurn := GC_UNITS_BY_REV_DRIVE;
		gBlock[iIndexBlock].parameters.Motor.DriveUnit.ScrewPitch.GearBox := 10.0;
		gBlock[iIndexBlock].parameters.Motor.DriveUnit.ScrewPitch.Pitch := 5.0;

		gBlock[iIndexBlock].parameters.Motor.rReferencePosition		:= 11.5;

		//Current Parameters
		gBlock[iIndexBlock].parameters.Motor.uiMaxCurrentBarsUp		:= 3;
		gBlock[iIndexBlock].parameters.Motor.uiMaxCurrentBarsDown		:= 1;

		gBlock[iIndexBlock].parameters.Motor.VerticalDirection:= MOTOR_POSITIVE;

		gBlock[iIndexBlock].parameters.Motor.rAcceleration		:= 172.5;
		gBlock[iIndexBlock].parameters.Motor.rDeceleration		:= 172.5;

		gBlock[iIndexBlock].parameters.Icla.DriveUnit.TransmissionType:=TRANS_LINEAL_PERIMETER;
		gBlock[iIndexBlock].parameters.Icla.DriveUnit.LinealPerimeter.GearBox:=92;
		gBlock[iIndexBlock].parameters.Icla.DriveUnit.LinealPerimeter.Perimeter:=180;
		gBlock[iIndexBlock].parameters.Icla.DriveUnit.LinealPerimeter.PulsesPerTurn:=12;

		gBlock[iIndexBlock].parameters.Inks.iMaxMachinePrintBars	:= 2;
		gBlock[iIndexBlock].parameters.Inks.iMaxBlockPrintBars		:= 2;
		gBlock[iIndexBlock].parameters.Inks.iMaxPSUwattsForBars		:= 3000;

		gBlock[iIndexBlock].parameters.xCappingProcess := FALSE;

		gBlock[iIndexBlock].parameters.Hw.SafetySignals := SAFETY_ESTOP_CALCULATED;

		//[RGP] Due to issue SUSTPLATF-236
		gBlock[iIndexBlock].parameters.xMotorOffsetAllowed := FALSE;

		gBlock[iIndexBlock].parameters.iApplicationBars := 2;
	END_FOR

	///////////////////////////////////////////////////
	/////PHOTOCELLS		PHOTOCELLS		 PHOTOCELLS////
	///////////////////////////////////////////////////

	gPhotoCells.parameters.xInstall := TRUE;
	gMachine.parSw.Hw.xInstallnSensor := FALSE;
	gPhotoCells.parameters.xSensorsPosHybridBehaviour := FALSE;

	gPhotoCells.parameters.MotorType := STP_STEPPER;
	gPhotoCells.parameters.AlignmentProcess := STP_ALIGNMENT_NO_REQUIRED;

	gPhotoCells.parameters.Speed:=2.5;
	gPhotoCells.parameters.JogSpeed:=1;
	gPhotoCells.parameters.Acceleration:=5;

	gPhotoCells.parameters.DriveUnit.TransmissionType := TRANS_SCREW_PITCH;
	gPhotoCells.parameters.DriveUnit.ScrewPitch.PulsesPerTurn := GC_UNITS_BY_REV_DRIVE;
	gPhotoCells.parameters.DriveUnit.ScrewPitch.GearBox := 1;
	gPhotoCells.parameters.DriveUnit.ScrewPitch.Pitch := 2.5;

	IF gMachine.Pt.ConfigNameID = GC_CONFIG_SIMTEST_ID THEN
		// In Simulation
		gPhotoCells.parameters.IndexDriveMaster:=4;
		gPhotoCells.parameters.IndexDriveSecondary:=5;
	ELSE
		gPhotoCells.parameters.IndexDriveMaster:=3;
		gPhotoCells.parameters.IndexDriveSecondary:=4;
	END_IF

	gPhotoCells.parameters.iSensorQuantity := 3;
	gPhotoCells.parameters.iSensorToReference := 2;
	gPhotoCells.parameters.rOffsetPosition := 0.0;
	gPhotoCells.parameters.rSensorMechPositionByPass := 65.0; //ALX -> ToReview
	gPhotoCells.parameters.Sensors[2].rDistanceRelativeToFirstSensor := 4;
	gPhotoCells.parameters.Sensors[3].rDistanceRelativeToFirstSensor := 8;
	gPhotoCells.parameters.xEnableMountedAlrByPass := TRUE;

	//Digital Inputs
	gPhotoCells.Inputs.Signals.pInput[1]	:= ADR (X1.DInput[1]);
	gPhotoCells.Inputs.Signals.pInput[2]	:= ADR (X1.DInput[2]);
	gPhotoCells.Inputs.Signals.pInput[3]	:= ADR (X1.DInput[3]);
	gPhotoCells.Inputs.Signals.xSafetyEnable := gMachine.In.xSafetyEnabled;

	stepperMotor ACCESS ADR (gAxis[gPhotoCells.parameters.IndexDriveMaster]);
	stepperMotor.Parameter.Direction:= MOTOR_NEGATIVE_AXIS;

	///////////////////////////////////////////////////
	/////DING			DING		DING	  DING/////
	///////////////////////////////////////////////////
	gDing.Parameters.xDingInstalled := FALSE;

	///////////////////////////////////////////////////
	/////THICKNESS		THICKNESS		 THICKNESS/////
	///////////////////////////////////////////////////

	//Configuring machine transport because some values are different in two blocks
	CASE gMachine.Pt.MachineModel OF
		Type_SHLD:
			gThicknessCtrl.parameters.iTotalBlocksLengh := 130;
			gThicknessCtrl.parameters.Belt.iDistanceEmptyBeltIni := 240;
		Type_SHLD_L:
			gThicknessCtrl.parameters.iTotalBlocksLengh := 130;
			gThicknessCtrl.parameters.Belt.iDistanceEmptyBeltIni := 390;
	END_CASE

	gThicknessCtrl.parameters.xMarginForBendTile := TRUE;
	gThicknessCtrl.parameters.rSafetyMarginToHeight := 3.0;

	gThicknessCtrl.parameters.sections[1].xEnabled	:= TRUE;
	gThicknessCtrl.parameters.sections[1].iStart	:= 1;
	gThicknessCtrl.parameters.sections[1].iEnd		:= 130;

	gThicknessCtrl.parameters.Detection.ProductDetect.xLoadMedia := FALSE;
	gThicknessCtrl.parameters.Detection.ProductDetect.iSensorPosition := 25;
	gThicknessCtrl.parameters.Detection.Analog.xLoadMedia := TRUE;
	gThicknessCtrl.parameters.Detection.Analog.iSensorPosition := 0;
	gThicknessCtrl.parameters.Detection.Array.xLoadMedia := TRUE;
	gThicknessCtrl.parameters.Detection.Array.iSensorPosition := 0;

	/////////////////////////////////////////////////////
	/////   TRANSPORT_VACUUM  TRANSPORT_VACUUM   ////////
	/////////////////////////////////////////////////////
	gTransVacuum[1].Parameters.xInstalled := FALSE;
	gTransVacuum[2].Parameters.xInstalled := FALSE;

	/////////////////////////////////////////////////////
	/////   NON_CRASH    NON_CRASH    NON_CRASH  ////////
	/////////////////////////////////////////////////////
	gNonCrash[1].Parameters.xInstalled := FALSE;

	/////////////////////////////////////////////////////
	/////   CHILLER 	CHILLER 	CHILLER 	/////////
	/////////////////////////////////////////////////////
	gMachine.Pt.Hw.iMaxNumChillers:=1;
	gChiller[1].Parameters.xInstalled := TRUE;
	gChiller[1].Parameters.SystemType := CHILLERSYS_WATERMANIFOLD;

	FOR iIndexInks:=1 TO MAX_LAST_INK DO
		gInks[iIndexInks].parameters.InksChiller.iIndex:=1;
	END_FOR

	// Always the last BLOCK of code
	/////////////////////////////////////////////////////
	/////   PLC CARDS	PLC CARDS	PLC CARDS	 ////////
	/////////////////////////////////////////////////////
	IF gPlcCards[0].Type <> CARD_UNDEFINED THEN
		RETURN;
	END_IF

	//Force "ModuleOk" in cards without it
	X20CPUData.ModuleOk := TRUE;
	X1.ModuleOk := TRUE;
	X2.ModuleOk := TRUE;
	X3.ModuleOk := TRUE;

	AsignCardsSHLD;

END_ACTION

ACTION AsignCardsSHLD:

	gPlcCards[0].Type := CARD_CPU1382;
	gPlcCards[0].pCard := ADR(X20CPUData);
	gPlcCards[0].RequiredForFunctions[0] := CARDREQUIRED_ALWAYS;
	gPlcCards[0].stCardName := 'X20CP1382_000';
	gPlcCards[0].Location := CardInPrinter;

	iIndexPlcCar := 1;
	// CARD 1 X1
	gPlcCards[iIndexPlcCar].Type := CARD_X1;
	gPlcCards[iIndexPlcCar].pCard := ADR(X1);
	gPlcCards[iIndexPlcCar].RequiredForFunctions[0] := CARDREQUIRED_ALWAYS;
	gPlcCards[iIndexPlcCar].stCardName := 'X2CP1382-X1_5N1';
	gPlcCards[iIndexPlcCar].Texts[1].Details := 'Spare';
	gPlcCards[iIndexPlcCar].Texts[2].Details := '';
	gPlcCards[iIndexPlcCar].Texts[3].Details := 'Spare';
	gPlcCards[iIndexPlcCar].Texts[4].Details := '';
	gPlcCards[iIndexPlcCar].Texts[5].Details := '';
	gPlcCards[iIndexPlcCar].Texts[6].Details := '';
	gPlcCards[iIndexPlcCar].Texts[7].Details := '3L-Detected tile(Phtcll 1)';
	gPlcCards[iIndexPlcCar].Texts[8].Details := '3L-Belt tile(Phtcll 2)';
	gPlcCards[iIndexPlcCar].Texts[9].Details := '3L-Mounted tile(Phtcll 3)';
	gPlcCards[iIndexPlcCar].Texts[10].Details := 'Bars ref. sensor-ON signa';
	gPlcCards[iIndexPlcCar].Texts[11].Details := 'CAN H';
	gPlcCards[iIndexPlcCar].Texts[12].Details := 'RS232 TXD';
	gPlcCards[iIndexPlcCar].Texts[13].Details := 'CAN L';
	gPlcCards[iIndexPlcCar].Texts[14].Details := 'RS232 RXD';
	gPlcCards[iIndexPlcCar].Texts[15].Details := 'GND';
	gPlcCards[iIndexPlcCar].Texts[16].Details := 'GND';
	gPlcCards[iIndexPlcCar].Location := CardInPrinter;
	iIndexPlcCar := iIndexPlcCar + 1;

	//CARD 2 X2
	gPlcCards[iIndexPlcCar].Type := CARD_X2;
	gPlcCards[iIndexPlcCar].pCard := ADR(X2);
	gPlcCards[iIndexPlcCar].RequiredForFunctions[0] := CARDREQUIRED_ALWAYS;
	gPlcCards[iIndexPlcCar].stCardName := 'X2CP1382-X2_5N1';
	gPlcCards[iIndexPlcCar].Texts[1].Details := '0Q21-Alarm(Transp. Driver)';
	gPlcCards[iIndexPlcCar].Texts[2].Details := '2Q35-Alarm(Elev. Driver)';
	gPlcCards[iIndexPlcCar].Texts[3].Details := '0D10-Alarm(48 VDC PH PSU)';
	gPlcCards[iIndexPlcCar].Texts[4].Details := '3T1-Thermostat alarm';
	gPlcCards[iIndexPlcCar].Texts[5].Details := 'PD-Broken sensor alarm';
	gPlcCards[iIndexPlcCar].Texts[6].Details := 'DPT-Broken sensor alarm';
	gPlcCards[iIndexPlcCar].Texts[7].Details := 'UPS-Failure UPS';
	gPlcCards[iIndexPlcCar].Texts[8].Details := 'UPS-Utility Failure';
	gPlcCards[iIndexPlcCar].Texts[9].Details := 'UPS-Low Battery';
	gPlcCards[iIndexPlcCar].Texts[10].Details := 'UPS-Inverter Failure';
	gPlcCards[iIndexPlcCar].Texts[11].Details := 'Spare';
	gPlcCards[iIndexPlcCar].Texts[12].Details := 'Spare';
	gPlcCards[iIndexPlcCar].Texts[13].Details := 'Spare';
	gPlcCards[iIndexPlcCar].Texts[14].Details := 'Spare';
	gPlcCards[iIndexPlcCar].Texts[15].Details := 'Spare';
	gPlcCards[iIndexPlcCar].Texts[16].Details := 'Spare';
	gPlcCards[iIndexPlcCar].Location := CardInPrinter;
	iIndexPlcCar := iIndexPlcCar + 1;

	//CARD 3 X3
	gPlcCards[iIndexPlcCar].Type := CARD_X3;
	gPlcCards[iIndexPlcCar].pCard := ADR(X3);
	gPlcCards[iIndexPlcCar].RequiredForFunctions[0] := CARDREQUIRED_ALWAYS;
	gPlcCards[iIndexPlcCar].stCardName := 'X2CP1382-X3_5N1';
	gPlcCards[iIndexPlcCar].Texts[1].Details := 'Spare';
	gPlcCards[iIndexPlcCar].Texts[2].Details := 'PC start from PLC';
	gPlcCards[iIndexPlcCar].Texts[3].Details := 'Reset Carriage Board';
	gPlcCards[iIndexPlcCar].Texts[4].Details := 'Reset Route';
	gPlcCards[iIndexPlcCar].Texts[5].Details := 'Spare';
	gPlcCards[iIndexPlcCar].Texts[6].Details := 'Spare';
	gPlcCards[iIndexPlcCar].Texts[7].Details := 'Spare';
	gPlcCards[iIndexPlcCar].Texts[8].Details := 'Spare';
	gPlcCards[iIndexPlcCar].Texts[9].Details := 'Spare';
	gPlcCards[iIndexPlcCar].Texts[10].Details := 'Spare';
	gPlcCards[iIndexPlcCar].Texts[11].Details := 'Spare';
	gPlcCards[iIndexPlcCar].Texts[12].Details := 'Spare';
	gPlcCards[iIndexPlcCar].Texts[13].Details := '+24VDC CPU/X2X';
	gPlcCards[iIndexPlcCar].Texts[14].Details := '+24VDC I/O';
	gPlcCards[iIndexPlcCar].Texts[15].Details := 'GND';
	gPlcCards[iIndexPlcCar].Texts[16].Details := 'GND';
	gPlcCards[iIndexPlcCar].Location := CardInPrinter;
	iIndexPlcCar := iIndexPlcCar + 1;

	//CARD 4 Digital Input
	gPlcCards[iIndexPlcCar].Type := CARD_DI16;
	gPlcCards[iIndexPlcCar].pCard := ADR(X20DIF371_001);
	gPlcCards[iIndexPlcCar].RequiredForFunctions[0] := CARDREQUIRED_ALWAYS;
	gPlcCards[iIndexPlcCar].stCardName := 'X20DIF371_001';
	gPlcCards[iIndexPlcCar].Texts[1].Details := 'Bar A Klixon';
	gPlcCards[iIndexPlcCar].Texts[2].Details := 'Bar B Klixon';
	gPlcCards[iIndexPlcCar].Texts[3].Details := 'Tank A - Empty Level';
	gPlcCards[iIndexPlcCar].Texts[4].Details := 'Tank B - Empty Level';
	gPlcCards[iIndexPlcCar].Texts[5].Details := 'Tank A - Full Level';
	gPlcCards[iIndexPlcCar].Texts[6].Details := 'Tank B - Full Level';
	gPlcCards[iIndexPlcCar].Texts[7].Details := 'Tank A - Presure Switch';
	gPlcCards[iIndexPlcCar].Texts[8].Details := 'Tank B - Presure Switch';
	gPlcCards[iIndexPlcCar].Texts[9].Details := 'Spare';
	gPlcCards[iIndexPlcCar].Texts[10].Details := 'Spare';
	gPlcCards[iIndexPlcCar].Texts[11].Details := 'Spare';
	gPlcCards[iIndexPlcCar].Texts[12].Details := 'Spare';
	gPlcCards[iIndexPlcCar].Texts[13].Details := 'Spare';
	gPlcCards[iIndexPlcCar].Texts[14].Details := 'Bars heater - 48VDC PSU OK';
	gPlcCards[iIndexPlcCar].Texts[15].Details := 'Bar A - 48VDC PSU OK';
	gPlcCards[iIndexPlcCar].Texts[16].Details := 'Bar B - 48VDC PSU OK';
	gPlcCards[iIndexPlcCar].Location := CardInPrinter;
	iIndexPlcCar := iIndexPlcCar + 1;

	//CARD 5 Digital Input
	gPlcCards[iIndexPlcCar].Type := CARD_DI16;
	gPlcCards[iIndexPlcCar].pCard := ADR(X20DIF371_002);
	gPlcCards[iIndexPlcCar].RequiredForFunctions[0] := CARDREQUIRED_ALWAYS;
	gPlcCards[iIndexPlcCar].stCardName := 'X20DIF371_002';
	gPlcCards[iIndexPlcCar].Texts[1].Details := 'Consents Line - Machine 1';
	gPlcCards[iIndexPlcCar].Texts[2].Details := 'Consents Line - Machine 2';
	gPlcCards[iIndexPlcCar].Texts[3].Details := 'Printhead External Cleaning';
	gPlcCards[iIndexPlcCar].Texts[4].Details := 'Spare';
	gPlcCards[iIndexPlcCar].Texts[5].Details := 'Start';
	gPlcCards[iIndexPlcCar].Texts[6].Details := 'Stop';
	gPlcCards[iIndexPlcCar].Texts[7].Details := 'Automatic';
	gPlcCards[iIndexPlcCar].Texts[8].Details := 'Zero';
	gPlcCards[iIndexPlcCar].Texts[9].Details := 'Manual';
	gPlcCards[iIndexPlcCar].Texts[10].Details := 'Validation to PLC';
	gPlcCards[iIndexPlcCar].Texts[11].Details := 'Machine confg. - Bit 1';
	gPlcCards[iIndexPlcCar].Texts[12].Details := 'Machine config. - Bit 2';
	gPlcCards[iIndexPlcCar].Texts[13].Details := 'Machine config. - Bit 3';
	gPlcCards[iIndexPlcCar].Texts[14].Details := 'Machine config. - Bit 4';
	gPlcCards[iIndexPlcCar].Texts[15].Details := 'Spare';
	gPlcCards[iIndexPlcCar].Texts[16].Details := 'Spare';
	gPlcCards[iIndexPlcCar].Location := CardInPrinter;
	iIndexPlcCar := iIndexPlcCar + 1;

	//CARD 6 Digital Input
	gPlcCards[iIndexPlcCar].Type := CARD_DI16;
	gPlcCards[iIndexPlcCar].pCard := ADR(X20DIF371_003);
	gPlcCards[iIndexPlcCar].RequiredForFunctions[0] := CARDREQUIRED_ALWAYS;
	gPlcCards[iIndexPlcCar].stCardName := 'X20DIF371_003';
	gPlcCards[iIndexPlcCar].Texts[1].Details := 'CB to PLC - Print trigger L2';
	gPlcCards[iIndexPlcCar].Texts[2].Details := 'CB to PLC - Print trigger L1';
	gPlcCards[iIndexPlcCar].Texts[3].Details := 'Spare';
	gPlcCards[iIndexPlcCar].Texts[4].Details := 'PC2 OK';
	gPlcCards[iIndexPlcCar].Texts[5].Details := 'Spare';
	gPlcCards[iIndexPlcCar].Texts[6].Details := 'Spare';
	gPlcCards[iIndexPlcCar].Texts[7].Details := 'Spare';
	gPlcCards[iIndexPlcCar].Texts[8].Details := 'Spare';
	gPlcCards[iIndexPlcCar].Texts[9].Details := 'Spare';
	gPlcCards[iIndexPlcCar].Texts[10].Details := 'Spare';
	gPlcCards[iIndexPlcCar].Texts[11].Details := 'Spare';
	gPlcCards[iIndexPlcCar].Texts[12].Details := 'Spare';
	gPlcCards[iIndexPlcCar].Texts[13].Details := 'Spare';
	gPlcCards[iIndexPlcCar].Texts[14].Details := 'Spare';
	gPlcCards[iIndexPlcCar].Texts[15].Details := 'Spare';
	gPlcCards[iIndexPlcCar].Texts[16].Details := 'Spare';
	gPlcCards[iIndexPlcCar].Location := CardInPrinter;
	iIndexPlcCar := iIndexPlcCar + 1;

	//CARD 7 Digital Input
	gPlcCards[iIndexPlcCar].Type := CARD_DI16;
	gPlcCards[iIndexPlcCar].pCard := ADR(X20DIF371_004);
	gPlcCards[iIndexPlcCar].RequiredForFunctions[0] := CARDREQUIRED_ALWAYS;
	gPlcCards[iIndexPlcCar].stCardName := 'X20DIF371_004';
	gPlcCards[iIndexPlcCar].Texts[1].Details := 'Chiller - Run OK';
	gPlcCards[iIndexPlcCar].Texts[2].Details := 'Chiller - General alarm';
	gPlcCards[iIndexPlcCar].Texts[3].Details := 'Water clean-Level sensor';
	gPlcCards[iIndexPlcCar].Texts[4].Details := 'Water clean-Pressure sensor';
	gPlcCards[iIndexPlcCar].Texts[5].Details := 'Spare';
	gPlcCards[iIndexPlcCar].Texts[6].Details := 'Spare';
	gPlcCards[iIndexPlcCar].Texts[7].Details := 'Spare';
	gPlcCards[iIndexPlcCar].Texts[8].Details := 'Spare';
	gPlcCards[iIndexPlcCar].Texts[9].Details := 'Safety module OK';
	gPlcCards[iIndexPlcCar].Texts[10].Details := 'Front Safety Switch-Alarm';
	gPlcCards[iIndexPlcCar].Texts[11].Details := 'Back Safety Switch-Alarm';
	gPlcCards[iIndexPlcCar].Texts[12].Details := 'Spare';
	gPlcCards[iIndexPlcCar].Texts[13].Details := 'Spare';
	gPlcCards[iIndexPlcCar].Texts[14].Details := 'Spare';
	gPlcCards[iIndexPlcCar].Texts[15].Details := 'Spare';
	gPlcCards[iIndexPlcCar].Texts[16].Details := 'Spare';
	gPlcCards[iIndexPlcCar].Location := CardInPrinter;
	iIndexPlcCar := iIndexPlcCar + 1;

	//CARD 8 Digital Output
	gPlcCards[iIndexPlcCar].Type := CARD_DO16;
	gPlcCards[iIndexPlcCar].pCard := ADR(X20DOF322_005);
	gPlcCards[iIndexPlcCar].RequiredForFunctions[0] := CARDREQUIRED_ALWAYS;
	gPlcCards[iIndexPlcCar].stCardName := 'X20DOF322_005';
	gPlcCards[iIndexPlcCar].Texts[1].Details := 'Bar A - 48 VDC PH PSU ON';
	gPlcCards[iIndexPlcCar].Texts[2].Details := 'Bar B - 48 VDC PH PSU ON';
	gPlcCards[iIndexPlcCar].Texts[3].Details := 'Bar A - Heating ON';
	gPlcCards[iIndexPlcCar].Texts[4].Details := 'Bar B - Heating ON';
	gPlcCards[iIndexPlcCar].Texts[5].Details := 'Bar A - Reverse _Solenoid 1 - 4';
	gPlcCards[iIndexPlcCar].Texts[6].Details := 'Bar B - Reverse _Solenoid 1 - 4';
	gPlcCards[iIndexPlcCar].Texts[7].Details := 'Bar A - Reverse _Solenoid 2 - 3';
	gPlcCards[iIndexPlcCar].Texts[8].Details := 'Bar B - Reverse _Solenoid 2 - 3';
	gPlcCards[iIndexPlcCar].Texts[9].Details := 'Bar A - Manifold tank EV';
	gPlcCards[iIndexPlcCar].Texts[10].Details := 'Bar B - Manifold tank EV';
	gPlcCards[iIndexPlcCar].Texts[11].Details := 'Spare';
	gPlcCards[iIndexPlcCar].Texts[12].Details := 'Chiller - Start';
	gPlcCards[iIndexPlcCar].Texts[13].Details := 'Cooling unit - Start';
	gPlcCards[iIndexPlcCar].Texts[14].Details := 'DTP Enable';
	gPlcCards[iIndexPlcCar].Texts[15].Details := 'PLC to CB - Simulation PD1';
	gPlcCards[iIndexPlcCar].Texts[16].Details := 'PLC to CB - Simulation PD2';
	gPlcCards[iIndexPlcCar].Location := CardInPrinter;
	iIndexPlcCar := iIndexPlcCar + 1;

	//CARD 9 Digital Output
	gPlcCards[iIndexPlcCar].Type := CARD_DO16;
	gPlcCards[iIndexPlcCar].pCard := ADR(X20DOF322_006);
	gPlcCards[iIndexPlcCar].RequiredForFunctions[0] := CARDREQUIRED_ALWAYS;
	gPlcCards[iIndexPlcCar].stCardName := 'X20DOF322_006';
	gPlcCards[iIndexPlcCar].Texts[1].Details := 'Consent - Line 1';
	gPlcCards[iIndexPlcCar].Texts[2].Details := 'Consent - Line 2';
	gPlcCards[iIndexPlcCar].Texts[3].Details := 'Compenser Line 1';
	gPlcCards[iIndexPlcCar].Texts[4].Details := 'Compenser Line 2';
	gPlcCards[iIndexPlcCar].Texts[5].Details := 'Warning Machine(Yellow)';
	gPlcCards[iIndexPlcCar].Texts[6].Details := 'Emergency Status(Red)';
	gPlcCards[iIndexPlcCar].Texts[7].Details := 'Line 1 - Ready Clean Up';
	gPlcCards[iIndexPlcCar].Texts[8].Details := 'Line 2 - Ready Clean Up';
	gPlcCards[iIndexPlcCar].Texts[9].Details := 'Suction Turbine';
	gPlcCards[iIndexPlcCar].Texts[10].Details := 'Spare';
	gPlcCards[iIndexPlcCar].Texts[11].Details := 'Spare';
	gPlcCards[iIndexPlcCar].Texts[12].Details := 'Status PLC-Run';
	gPlcCards[iIndexPlcCar].Texts[13].Details := 'Zero mode-Air supply off';
	gPlcCards[iIndexPlcCar].Texts[14].Details := 'Start Green Light ON';
	gPlcCards[iIndexPlcCar].Texts[15].Details := 'Reset blue light ON';
	gPlcCards[iIndexPlcCar].Texts[16].Details := 'Buzzer';
	gPlcCards[iIndexPlcCar].Location := CardInPrinter;
	iIndexPlcCar := iIndexPlcCar + 1;

	//CARD 10 Power Supply
	gPlcCards[iIndexPlcCar].Type := CARD_PS33;
	gPlcCards[iIndexPlcCar].pCard := ADR(X20PS3300_007);
	gPlcCards[iIndexPlcCar].RequiredForFunctions[0] := CARDREQUIRED_ALWAYS;
	gPlcCards[iIndexPlcCar].stCardName := 'X20PS3300_007';
	gPlcCards[iIndexPlcCar].Location := CardInPrinter;
	iIndexPlcCar := iIndexPlcCar + 1;

	//CARD 11 Analog Input
	gPlcCards[iIndexPlcCar].Type := CARD_AI4;
	gPlcCards[iIndexPlcCar].pCard := ADR(X20AI4322_008);
	gPlcCards[iIndexPlcCar].RequiredForFunctions[0] := CARDREQUIRED_ALWAYS;
	gPlcCards[iIndexPlcCar].stCardName := 'X20AI4322_008';
	gPlcCards[iIndexPlcCar].Texts[1].Details := 'BarA-Pos Manifold Pres. Sensor';
	gPlcCards[iIndexPlcCar].Texts[2].Details := 'BarB-Pos Manifold Pres. Sensor';
	gPlcCards[iIndexPlcCar].Texts[3].Details := 'BarA-Neg Manifold Pres. Sensor';
	gPlcCards[iIndexPlcCar].Texts[4].Details := 'BarB-Neg Manifold Pres. Sensor';
	gPlcCards[iIndexPlcCar].Location := CardInPrinter;
	iIndexPlcCar := iIndexPlcCar + 1;

	//CARD 12 Analog Output
	gPlcCards[iIndexPlcCar].Type := CARD_AO4;
	gPlcCards[iIndexPlcCar].pCard := ADR(X20AO4622_009);
	gPlcCards[iIndexPlcCar].RequiredForFunctions[0] := CARDREQUIRED_ALWAYS;
	gPlcCards[iIndexPlcCar].stCardName := 'X20AO4622_009';
	gPlcCards[iIndexPlcCar].Texts[1].Details := 'BarA - Pump';
	gPlcCards[iIndexPlcCar].Texts[2].Details := 'BarB - Pump';
	gPlcCards[iIndexPlcCar].Texts[3].Details := 'TankA - Pump';
	gPlcCards[iIndexPlcCar].Texts[4].Details := 'TankB - Pump';
	gPlcCards[iIndexPlcCar].Location := CardInPrinter;
	iIndexPlcCar := iIndexPlcCar + 1;

	//CARD 13 Analog Input
	gPlcCards[iIndexPlcCar].Type := CARD_AT4;
	gPlcCards[iIndexPlcCar].pCard := ADR(X20AT4222_010);
	gPlcCards[iIndexPlcCar].RequiredForFunctions[0] := CARDREQUIRED_ALWAYS;
	gPlcCards[iIndexPlcCar].stCardName := 'X20AT4222_010';
	gPlcCards[iIndexPlcCar].Texts[1].Details := 'BarA - Temp Probe (Manifold)';
	gPlcCards[iIndexPlcCar].Texts[2].Details := 'BarB - Temp Probe (Manifold)';
	gPlcCards[iIndexPlcCar].Texts[3].Details := 'Chiller - Tank cabinet temp PT100';
	gPlcCards[iIndexPlcCar].Texts[4].Details := 'Chiller - In water temp PT100';
	gPlcCards[iIndexPlcCar].Location := CardInPrinter;
	iIndexPlcCar := iIndexPlcCar + 1;

	//CARD 14 Stepper Driver
	gPlcCards[iIndexPlcCar].Type := CARD_SM;
	gPlcCards[iIndexPlcCar].pCard := ADR(X20SM1436_011);
	gPlcCards[iIndexPlcCar].RequiredForFunctions[0] := CARDREQUIRED_ALWAYS;
	gPlcCards[iIndexPlcCar].stCardName := 'X20SM1436_011';
	gPlcCards[iIndexPlcCar].Location := CardInPrinter;
	iIndexPlcCar := iIndexPlcCar + 1;

	//CARD 15 Stepper Driver
	gPlcCards[iIndexPlcCar].Type := CARD_SM;
	gPlcCards[iIndexPlcCar].pCard := ADR(X20SM1436_012);
	gPlcCards[iIndexPlcCar].RequiredForFunctions[0] := CARDREQUIRED_ALWAYS;
	gPlcCards[iIndexPlcCar].stCardName := 'X20SM1436_012';
	gPlcCards[iIndexPlcCar].Location := CardInPrinter;
	iIndexPlcCar := iIndexPlcCar + 1;

	//END CARDS

	gPlcCards[iIndexPlcCar].Type := CARD_UNDEFINED;

END_ACTION
```

#### AssignDataMecano.st
```iecst
ACTION AssignDataMecano:

	//Just writing the fixed configuration once per each 5s
	IF gMachine.Pt.ConfigNameID <> GC_CONFIG_PLCDIAGNOSIS_ID AND NOT (EDGEPOS(gPLC.xBlk_5s) OR gPLC.xFirst_Scan OR xChangedSimMachine) THEN
		RETURN;
	END_IF

	////////////////////////////////////////////////////////////
	/////GENERAL	GENERAL		GENERAL		GENERAL	////////////
	////////////////////////////////////////////////////////////
	gMachine.Pt.xControlledRemotely := FALSE;
	gMachine.Pt.xDisableStartHoldingGreenButton := TRUE;

	gMachine.Pt.CT.rMountedMediaLevelInBypassMode		:= 145.0;
	gMachine.Pt.CT.rMaxTicknessMedia		:= 30.0;
	gMachine.Pt.CT.rMinTicknessMedia		:= 0.3;
	gMachine.Pt.CT.iNumSAIInstalled			:= 2;
	gMachine.Pt.CT.rDistanceThicknesToPD	:= 203.8;
	gMachine.Pt.CT.rDistanceBeltInitToPd	:= 2400; //To review

	gMachine.Pt.rMaxPrintHeadPos			:= 1900.0;
	gMachine.Pt.rMinPrintHeadPos			:= 10;
	gMachine.Pt.CT.rMinMarginPrinting		:= 1.7;
	gMachine.Pt.rBeltSpeedWhileEmptyBelt	:= 20.0; //m/min

	gMachine.Pt.iMediaFilter 				:= 20;

	gMachine.parSw.rFirstHeadPosition 		:= 30.0; //[RGP] This parameter should not be written here. To remove after SW release
	gMachine.parSw.rLastHeadPosition 		:= 1870; //[RGP] This parameter should not be written here. To remove after SW release
	gMachine.parSw.xJamDetectEnable			:= TRUE; //DELOREAN-1031 //[RGP] To discuss internally with plc team why is optional for BM machines and not for Nz2

	gMachine.Pt.PDSignalTpe 						:= PDCFG_SENSOR;
	gMachine.Pt.xProtectPHWithStoppedMediaBended	:= FALSE;
	gMachine.Pt.xProtectPHForBlowersRunning			:= TRUE;
	gMachine.Pt.Clean.xCleanBeltTopInstall 			:= FALSE;
	gMachine.Pt.xAllowLaboratory	 				:= FALSE;
	gMachine.Pt.xAllowJamRecovery	 				:= FALSE;
	gMachine.Pt.xDynamicPrePrintingPos				:= TRUE;
	gMachine.Pt.xJobNotReadyIsCritical	 			:= TRUE;
	gMachine.Pt.Clean.xCleanBeltForUv 				:= FALSE; //Set to FALSE due to DELOREAN-3204 //gMachine.Pt.MachineModel <> Type_NOZ_2_AQ;
	gMachine.Pt.CommsType							:= Type_OpcUa;

	gMachine.Pt.Cure.xCuringByStretchAllowed := TRUE;

	gMachine.Pt.Hw.iWidth					:= 1700;
	gMachine.Pt.Hw.rMinPrintPosition		:= 2.0; //To review regarding SD requirements. Min thickness 0.3 and minimum jetting gap is 1.7, but may be changed in the future
	gMachine.Pt.Hw.xDoubleLineAllowed		:= FALSE;
	gMachine.Pt.Hw.xSuctionModeAllowed		:= TRUE;

	gMachine.St.HwData.xIsPlatform5			:= FALSE;
	gMachine.St.HwData.xIsWater				:= gMachine.Pt.MachineModel=Type_NOZ_2_AQ;
	gMachine.St.HwData.xIsCubik				:= FALSE;
	gMachine.St.HwData.xUpsOutOfPrinter		:= Pdc_X20DIF371_040.ModuleOk; //Codified card used when UPS are installed inside the PDC

	gMachine.St.White.xInstalled := FALSE;
	gMachine.St.Color.xInstalled := FALSE;
	gMachine.St.Clear.xInstalled := FALSE;
	FOR iIndexCuringLedLamps:=1 TO MAX_LAST_CURING_LED DO
		IF gCuringLed[iIndexCuringLedLamps].Parameters.CuringApplicationType = CURING_APP_WHITE THEN
			gMachine.St.White.xInstalled := TRUE;
		ELSIF gCuringLed[iIndexCuringLedLamps].Parameters.CuringApplicationType = CURING_APP_PRIMER THEN
			gMachine.St.Clear.xInstalled := TRUE;
		ELSIF gCuringLed[iIndexCuringLedLamps].Parameters.CuringApplicationType = CURING_APP_COLOR THEN
			gMachine.St.Color.xInstalled := TRUE;
		END_IF
	END_FOR

	//Belt
	gBelt.parameters.xRemoteAcceleration := FALSE;
	gBelt.parameters.xRemoteDeceleration := FALSE;
	gBelt.parameters.rAcceleration := 1050;
	gBelt.parameters.rDeceleration := 2400;
	gBelt.parameters.rMaxAcceleration := 1500.0;
	gBelt.parameters.rMaxDeceleration := 2500.0;

	//Here are configured blocks in function of the machine direction
	//When machine is block then we need use correction as block physical 2 because PD is at the same distance than Block 1, for that is change process in function of machine 2 Blcoks or machine 1 block
	gBlock[1].parameters.iMotorAxisIndex := 2;
	gBlock[1].parameters.iMappingBlock := 1;
	gBlock[1].parameters.iIclaAxisIndex := 1;
	gBlock[1].parameters.Hw.ValvesCommsType := COMMS_POWERLINK;
	gBlock[1].parSw.xEnableToMovements := TRUE; //[RGP] This parameter should not be written here. To remove after SW release
	gBlock[1].parSw.xEnableToPrint := TRUE; //[RGP] This parameter should not be written here. To remove after SW release

	gMachine.parSw.xMachineDirection := TRUE; //Machine from left //[RGP] This parameter should not be written here. To remove after SW release

	////////////////////////////////////////////////////////////
	/////BLOCK	BLOCK	BLOCK	BLOCK	BLOCK	BLOCK///////////
	////////////////////////////////////////////////////////////
	FOR iIndexBlock:=1 TO gMachine.Pt.CT.iNumBlocks DO

		//Position parameters (mm)
		gBlock[iIndexBlock].parameters.Motor.rSafePosition				:= 356.0;	//Max heigh
		gBlock[iIndexBlock].parameters.Motor.rMinSafePosition			:= 2.0;		//Min heigh
		gBlock[iIndexBlock].parameters.Motor.rCapPosition				:= 344.0;	//CAP
		gBlock[iIndexBlock].parameters.Motor.rCappingPosition			:= 251.0; 	//CAPPING
		gBlock[iIndexBlock].parameters.Motor.rSafePositionCleanCarrier	:= 329.0;	//Carrier out Safe
		gBlock[iIndexBlock].parameters.Motor.rDripBarsPosition			:= 279.0;	//Drip
		gBlock[iIndexBlock].parameters.Motor.rCleanPosition				:= 335.0; 	//Clean
		gBlock[iIndexBlock].parameters.Motor.rWaterSpurtPosition		:= 342.0;	//Water Spurt

		gBlock[iIndexBlock].parameters.Motor.rAutoSpeedMoveDown	:=30.0;
		gBlock[iIndexBlock].parameters.Motor.rAutoSpeedMoveUp	:=30.0;
		IF gMachine.Pt.ConfigNameID <> GC_CONFIG_SIMTEST_ID THEN
			gBlock[iIndexBlock].parameters.Motor.rAutoSpeedMoveUpFast	:= 50.0;
		ELSE
			gBlock[iIndexBlock].parameters.Motor.rAutoSpeedMoveUpFast	:= gBlock[iIndexBlock].parameters.Motor.rAutoSpeedMoveUp + 1; //Modifying value in sim just for testing purposes
		END_IF
		gBlock[iIndexBlock].parameters.Motor.xFastSpeedAllowed	:= TRUE;
		gBlock[iIndexBlock].parameters.Motor.xOversized	:= TRUE;
		gBlock[iIndexBlock].parameters.Motor.rOperationTorque	:= 10.0;
		gBlock[iIndexBlock].parameters.Motor.DriveUnit.TransmissionType := TRANS_SCREW_PITCH;
		gBlock[iIndexBlock].parameters.Motor.DriveUnit.ScrewPitch.PulsesPerTurn := GC_UNITS_BY_REV_DRIVE;
		gBlock[iIndexBlock].parameters.Motor.DriveUnit.ScrewPitch.GearBox := 5.2;
		gBlock[iIndexBlock].parameters.Motor.DriveUnit.ScrewPitch.Pitch := 5.0;

		gBlock[iIndexBlock].parameters.Motor.rReferencePosition			:= 15.5;

		//Current Parameters
		gBlock[iIndexBlock].parameters.Motor.uiMaxCurrentBarsUp			:= 3;
		gBlock[iIndexBlock].parameters.Motor.uiMaxCurrentBarsDown		:= 1;

		gBlock[iIndexBlock].parameters.Motor.VerticalDirection:= MOTOR_POSITIVE;

		gBlock[iIndexBlock].parameters.Motor.rAcceleration				:= 260;
		gBlock[iIndexBlock].parameters.Motor.rDeceleration				:= 260;

		gBlock[iIndexBlock].parameters.Icla.DriveUnit.TransmissionType:=TRANS_LINEAL_PERIMETER;
		gBlock[iIndexBlock].parameters.Icla.DriveUnit.LinealPerimeter.GearBox:=92;
		gBlock[iIndexBlock].parameters.Icla.DriveUnit.LinealPerimeter.Perimeter:=180;
		gBlock[iIndexBlock].parameters.Icla.DriveUnit.LinealPerimeter.PulsesPerTurn:=12;

		gBlock[iIndexBlock].parameters.Inks.iMaxMachinePrintBars	:= 7;
		gBlock[iIndexBlock].parameters.Inks.iMaxBlockPrintBars		:= 7;
		gBlock[iIndexBlock].parameters.Inks.iMaxPSUwattsForBars		:= 3000;

		gBlock[iIndexBlock].parameters.xCappingProcess := FALSE; // Capping hardware removed from 14000LED Bill of materials. Not removed from code, just disabled (Nozomi-2150) //Machine.Pt.MachineModel=Type_NOZ_2_AQ;
		gBlock[iIndexBlock].parameters.xWastedInkTankProcess := TRUE;

		gBlock[iIndexBlock].parameters.iFirstBarPosition := 50; //512mm measured in 3D model by mechanical team
		gBlock[iIndexBlock].parameters.iLastBarPosition := 480; //2462mm measured in 3D model by mechanical team for eight bar position. This parameters consider distance till end of bars block

		gBlock[iIndexBlock].parameters.Hw.SafetySignals := SAFETY_ESTOP_CONNECTED;

		//[RGP] Due to issue SUSTPLATF-236
		gBlock[iIndexBlock].parameters.xMotorOffsetAllowed := FALSE;

		gBlock[iIndexBlock].parameters.iApplicationBars := 9;
	END_FOR

	FOR iIndexInks:=1 TO MAX_LAST_INK DO
		//If not in debug mode, assign values because in this machine they have not UI interface
		IF NOT gInks[iIndexInks].parameters.xDebugMode THEN
			gInks[iIndexInks].parSw.NegPump.rUpperLimMeniscusCritical := 60.0;
			gInks[iIndexInks].parSw.NegPump.rLowerLimMeniscusCritical := -30.0; //0.0;
			gInks[iIndexInks].parSw.NegPump.rLimitMeniscusDiffWarning := 5.0;
		END_IF
	END_FOR

	///////////////////////////////////////////////////
	/////PHOTOCELLS		PHOTOCELLS		PHOTOCELLS/////
	///////////////////////////////////////////////////

	gPhotoCells.parameters.xInstall := TRUE;
	gMachine.parSw.Hw.xInstallnSensor := FALSE;
	gPhotoCells.parameters.xSensorsPosHybridBehaviour := TRUE;

	gPhotoCells.parameters.MotorType := STP_ICLA;
	gPhotoCells.parameters.AlignmentProcess := STP_ALIGNMENT_REQUIRED;

	gPhotoCells.parSw.rMechOffset := 0.0; //Forced here because this parameter is not allowed in this machine
	gPhotoCells.parameters.rDistanceBetweenSensors := 25;
	gPhotoCells.parameters.rSensorMechPositionMax := 75;
	gPhotoCells.parameters.rSensorTeoMechPositionAlignment := 68.4; //DELOREAN-3539
	gPhotoCells.parameters.rSensorMechPositionAlignmentMax := gPhotoCells.parameters.rSensorTeoMechPositionAlignment + gPhotoCells.parameters.rSensorMechToleranceAlignment;
	gPhotoCells.parameters.rSensorMechPositionAlignmentMin := gPhotoCells.parameters.rSensorTeoMechPositionAlignment - gPhotoCells.parameters.rSensorMechToleranceAlignment;

	gPhotoCells.parameters.Speed:=10;
	gPhotoCells.parameters.JogSpeed:= 10;
	gPhotoCells.parameters.Acceleration:=5;

	gPhotoCells.parameters.DriveUnit.TransmissionType := TRANS_SCREW_PITCH;
	gPhotoCells.parameters.DriveUnit.ScrewPitch.PulsesPerTurn := 12;
	gPhotoCells.parameters.DriveUnit.ScrewPitch.GearBox := 92;
	gPhotoCells.parameters.DriveUnit.ScrewPitch.Pitch := 4;

	IF gMachine.Pt.ConfigNameID = GC_CONFIG_SIMTEST_ID THEN
		// In Simulation
		gPhotoCells.parameters.IndexIcla:=3;
	ELSE
		gPhotoCells.parameters.IndexIcla:=2;
	END_IF

	gPhotoCells.parameters.iSensorQuantity := 6;
	gPhotoCells.parameters.iSensorToReference := 1;
	gPhotoCells.parameters.rOffsetPosition := -0.5;
	gPhotoCells.parameters.rOffsetRelToBar := 0.5;
	gPhotoCells.parameters.rSensorMechPositionByPass := 65;
	gPhotoCells.parameters.Sensors[2].rDistanceRelativeToFirstSensor := 1.5;
	gPhotoCells.parameters.Sensors[3].rDistanceRelativeToFirstSensor := 3;
	gPhotoCells.parameters.Sensors[4].rDistanceRelativeToFirstSensor := 4.5;
	gPhotoCells.parameters.Sensors[5].rDistanceRelativeToFirstSensor := 6;
	gPhotoCells.parSw.Sensors[5].xToRejectMedia := TRUE;
	gPhotoCells.parameters.Sensors[6].rDistanceRelativeToFirstSensor := 21;
	gPhotoCells.parameters.xEnableMountedAlrByPass := FALSE;

	///////////////////////////////////////////////////
	/////DING		DING		DING		DING  /////
	///////////////////////////////////////////////////
	gDing.Parameters.xDingInstalled := FALSE;

	///////////////////////////////////////////////////
	/////THICKNESS		THICKNESS		 THICKNESS/////
	///////////////////////////////////////////////////

	//Configuring machine transport because some values are different in two blocks
	gThicknessCtrl.parameters.xMarginForBendTile := FALSE;

	gThicknessCtrl.parameters.iTotalBlocksLengh := 305;
	gThicknessCtrl.parameters.Belt.iDistanceEmptyBeltIni := 470; //This distance is mechanical. Not related with Reject. Reject MUST not be eadjusted with this
	gThicknessCtrl.parameters.Belt.iBeltPerimeterLength := 1275;

	gThicknessCtrl.parameters.sections[1].xEnabled	:= TRUE;
	gThicknessCtrl.parameters.sections[1].iStart	:= 1;
	gThicknessCtrl.parameters.sections[1].iEnd		:= 500;

	gThicknessCtrl.parameters.Detection.ProductDetect.xLoadMedia := TRUE;
	gThicknessCtrl.parameters.Detection.ProductDetect.iSensorPosition := 20;
	gThicknessCtrl.parameters.Detection.Analog.xLoadMedia := FALSE;
	gThicknessCtrl.parameters.Detection.Analog.iSensorPosition := 0;
	gThicknessCtrl.parameters.Detection.Array.xLoadMedia := FALSE;
	gThicknessCtrl.parameters.Detection.Array.iSensorPosition := 0;

	gThicknessCtrl.parameters.Reject.xRejectTracking := TRUE;

	/////////////////////////////////////////////////////
	/////   TRANSPORT_VACUUM  TRANSPORT_VACUUM   ////////
	/////////////////////////////////////////////////////
	gMachine.Pt.Vacuum.xTransVacuumIndependenParams:=FALSE;

	gTransVacuum[1].Parameters.xInstalled := TRUE;
	gTransVacuum[1].Parameters.Hw.xSystemWithJoints := TRUE;
	gTransVacuum[1].Parameters.Hw.uiNumBlowers := 2;
	gTransVacuum[1].Parameters.Hw.BlowerData[1].iIndex := 1;
	gTransVacuum[1].Parameters.Hw.BlowerData[2].iIndex := 4;

	gTransVacuum[1].Parameters.Hw.BlowerData[1].Direction := MOTOR_NEGATIVE;
	gTransVacuum[1].Parameters.Hw.BlowerData[2].Direction := MOTOR_POSITIVE;

	gTransVacuum[1].Parameters.xStartUpEnable := FALSE;
	gTransVacuum[1].Parameters.rMinVacPressureSetPointPerc := 4.0;
	gTransVacuum[1].Parameters.rMinDutyCycle := 20.0;

	gTransVacuum[2].Parameters.xInstalled := TRUE;
	gTransVacuum[2].Parameters.Hw.xSystemWithJoints := TRUE;
	gTransVacuum[2].Parameters.Hw.uiNumBlowers := 2;
	gTransVacuum[2].Parameters.Hw.BlowerData[1].iIndex := 2;
	gTransVacuum[2].Parameters.Hw.BlowerData[2].iIndex := 3;
	gTransVacuum[2].Parameters.Hw.BlowerData[1].Direction := MOTOR_POSITIVE;
	gTransVacuum[2].Parameters.Hw.BlowerData[2].Direction := MOTOR_NEGATIVE;
	gTransVacuum[2].Parameters.xStartUpEnable := FALSE;
	gTransVacuum[2].Parameters.rMinVacPressureSetPointPerc := 4.0;
	gTransVacuum[2].Parameters.rMinDutyCycle := 20.0;

	FOR iIndexTrVacc := 1 TO MAX_LAST_TRANS_VACUUM DO
		gTransVacuum[iIndexTrVacc].Parameters.parPID.rKp := 0.4; //0.5;
		gTransVacuum[iIndexTrVacc].Parameters.parPID.rTi := 1.5;
		gTransVacuum[iIndexTrVacc].Parameters.parPID.rKd := 0.0;
		gTransVacuum[iIndexTrVacc].Parameters.parPID.rTd := 0.0;

		gTransVacuum[iIndexTrVacc].Parameters.rMaxSystemVacuum := 31.2; //DELOREAN-2860: Modified from 2400Pa to 3120Pa
		gTransVacuum[iIndexTrVacc].Parameters.rMaxSpeed := 3000;
		gTransVacuum[iIndexTrVacc].Parameters.rMaxPIDOut := 100.0;
	END_FOR

	// The rule for this parameter is (iTotalAreas -1) x rAreaWidth + rCentralAreaWithoutVacuum = vaccum width -> 17 x 68 + 495 = 1.651 distance from simetric max width slots
	gTransVacuum[1].Parameters.Hw.iTotalAreas := 18;
	gTransVacuum[1].Parameters.Hw.rAreaWidth := 68;
	gTransVacuum[1].Parameters.Hw.rCentralAreaWithoutVacuum := 495;

	/////////// CURING LED BARS ///////////
	iIndexWhiteCuringLedBar := 0;
	iIndexColorCuringLedBar := 0;
	iIndexPrimerCuringLedBar := 0;

	CASE gMachine.Pt.MachineModel OF

		Type_MECANO_UV_WHITE:
			gMachine.Pt.Hw.iMaxCuringLedBars := 2;
			IF gMachine.Pt.ConfigNameID <> GC_CONFIG_SIMTEST_ID THEN
				IF X20CS1030_180.ModuleOk THEN
					iIndexWhiteCuringLedBar := 1;
					iIndexColorCuringLedBar := 2;
				ELSE
					iIndexColorCuringLedBar := 1;
				END_IF

			ELSE
				iIndexWhiteCuringLedBar := 1;
				iIndexColorCuringLedBar := 2;
			END_IF

		Type_MECANO_UV_OPV:
			gMachine.Pt.Hw.iMaxCuringLedBars := 2;
			iIndexColorCuringLedBar := 1;
			IF X20CS1030_181.ModuleOk THEN
				iIndexPrimerCuringLedBar := 2;
			END_IF

		Type_MECANO_UV_WHITE_OPV:
			gMachine.Pt.Hw.iMaxCuringLedBars := 3;
			IF gMachine.Pt.ConfigNameID <> GC_CONFIG_SIMTEST_ID THEN
				IF X20CS1030_180.ModuleOk THEN
					iIndexWhiteCuringLedBar := 1;
					iIndexColorCuringLedBar := 2;
					IF X20CS1030_181.ModuleOk THEN
						iIndexPrimerCuringLedBar := 3;
					END_IF
				ELSE
					iIndexColorCuringLedBar := 1;
					IF X20CS1030_181.ModuleOk THEN
						iIndexPrimerCuringLedBar := 2;
					END_IF
				END_IF

			ELSE
				iIndexWhiteCuringLedBar := 1;
				iIndexColorCuringLedBar := 2;
				iIndexPrimerCuringLedBar := 3;
			END_IF

		END_CASE

	//Curing leds
	IF gMachine.Pt.ConfigNameID <> GC_CONFIG_SIMTEST_ID THEN
		gCuringLed[iIndexWhiteCuringLedBar].Parameters.xInstalled := X20CS1030_180.ModuleOk;
	ELSE
		gCuringLed[iIndexWhiteCuringLedBar].Parameters.xInstalled := (gMachine.Pt.MachineModel=Type_MECANO_UV_WHITE OR gMachine.Pt.MachineModel=Type_MECANO_UV_WHITE_OPV);
	END_IF
	gCuringLed[iIndexWhiteCuringLedBar].Parameters.iPowerSuppliesQuantity := 4;
	gCuringLed[iIndexWhiteCuringLedBar].Parameters.iLampsQuantity := 5;
	gCuringLed[iIndexWhiteCuringLedBar].Parameters.iCuringWindow := 40;
	gCuringLed[iIndexWhiteCuringLedBar].Parameters.rMinCureSpeed := 1;
	gCuringLed[iIndexWhiteCuringLedBar].Lamp[1].Parameters.iCuringLength := 350;
	gCuringLed[iIndexWhiteCuringLedBar].Lamp[2].Parameters.iCuringLength := 350;
	gCuringLed[iIndexWhiteCuringLedBar].Lamp[3].Parameters.iCuringLength := 350;
	gCuringLed[iIndexWhiteCuringLedBar].Lamp[4].Parameters.iCuringLength := 350;
	gCuringLed[iIndexWhiteCuringLedBar].Lamp[5].Parameters.iCuringLength := 350;
	gCuringLed[iIndexWhiteCuringLedBar].Parameters.iCuringPosition := 55;
	gCuringLed[iIndexWhiteCuringLedBar].Parameters.iChillerIndex := 2;
	gCuringLed[iIndexWhiteCuringLedBar].Parameters.CuringApplicationType := CURING_APP_WHITE;
	gCuringLed[iIndexWhiteCuringLedBar].Parameters.iMappingBar := 9;
	gCuringLed[iIndexWhiteCuringLedBar].Parameters.xPhysicalTempFeedback := FALSE;
	gCuringLed[iIndexWhiteCuringLedBar].Comms.Device.DeviceName := 'IF3.ST131.IF1.ST80.IF1';

	//OVCMYK curing led
	gCuringLed[iIndexColorCuringLedBar].Parameters.xInstalled := TRUE;
	gCuringLed[iIndexColorCuringLedBar].Parameters.iPowerSuppliesQuantity := 6;
	gCuringLed[iIndexColorCuringLedBar].Parameters.iLampsQuantity := 5;
	gCuringLed[iIndexColorCuringLedBar].Parameters.iCuringWindow := 80;
	gCuringLed[iIndexColorCuringLedBar].Parameters.rMinCureSpeed := 1;
	gCuringLed[iIndexColorCuringLedBar].Lamp[1].Parameters.iCuringLength := 350;
	gCuringLed[iIndexColorCuringLedBar].Lamp[2].Parameters.iCuringLength := 350;
	gCuringLed[iIndexColorCuringLedBar].Lamp[3].Parameters.iCuringLength := 350;
	gCuringLed[iIndexColorCuringLedBar].Lamp[4].Parameters.iCuringLength := 350;
	gCuringLed[iIndexColorCuringLedBar].Lamp[5].Parameters.iCuringLength := 350;
	gCuringLed[iIndexColorCuringLedBar].Parameters.iCuringPosition := 230;
	gCuringLed[iIndexColorCuringLedBar].Parameters.iChillerIndex := 1;
	gCuringLed[iIndexColorCuringLedBar].Parameters.CuringApplicationType := CURING_APP_COLOR;
	IF gMachine.Pt.MachineModel = Type_MECANO_UV_WHITE THEN
		gCuringLed[iIndexColorCuringLedBar].Parameters.iMappingBar := 2;
	ELSE
		gCuringLed[iIndexColorCuringLedBar].Parameters.iMappingBar := 4;
	END_IF
	gCuringLed[iIndexColorCuringLedBar].Parameters.xPhysicalTempFeedback := FALSE;
	gCuringLed[iIndexColorCuringLedBar].Comms.Device.DeviceName := 'IF3.ST131.IF1.ST62.IF1';

	//Primer curing led
	IF gMachine.Pt.ConfigNameID <> GC_CONFIG_SIMTEST_ID THEN
		gCuringLed[iIndexPrimerCuringLedBar].Parameters.xInstalled := X20CS1030_181.ModuleOk;
	ELSE
		gCuringLed[iIndexPrimerCuringLedBar].Parameters.xInstalled := FALSE; //(gMachine.Pt.MachineModel=Type_MECANO_UV_OPV OR gMachine.Pt.MachineModel=Type_MECANO_UV_WHITE_OPV);
	END_IF
	gCuringLed[iIndexPrimerCuringLedBar].Parameters.iPowerSuppliesQuantity := 6;
	gCuringLed[iIndexPrimerCuringLedBar].Parameters.iLampsQuantity := 5;
	gCuringLed[iIndexPrimerCuringLedBar].Parameters.iCuringWindow := 80;
	gCuringLed[iIndexPrimerCuringLedBar].Parameters.rMinCureSpeed := 1;
	gCuringLed[iIndexPrimerCuringLedBar].Lamp[1].Parameters.iCuringLength := 350;
	gCuringLed[iIndexPrimerCuringLedBar].Lamp[2].Parameters.iCuringLength := 350;
	gCuringLed[iIndexPrimerCuringLedBar].Lamp[3].Parameters.iCuringLength := 350;
	gCuringLed[iIndexPrimerCuringLedBar].Lamp[4].Parameters.iCuringLength := 350;
	gCuringLed[iIndexPrimerCuringLedBar].Lamp[5].Parameters.iCuringLength := 350;
	gCuringLed[iIndexPrimerCuringLedBar].Parameters.iCuringPosition := 290;
	gCuringLed[iIndexPrimerCuringLedBar].Parameters.iChillerIndex := 2;
	gCuringLed[iIndexPrimerCuringLedBar].Parameters.CuringApplicationType := CURING_APP_PRIMER;
	gCuringLed[iIndexPrimerCuringLedBar].Parameters.iMappingBar := 2;
	gCuringLed[iIndexPrimerCuringLedBar].Parameters.xPhysicalTempFeedback := FALSE;
	gCuringLed[iIndexPrimerCuringLedBar].Comms.Device.DeviceName := 'IF3.ST131.IF1.ST81.IF1';

	//CHILLER
	FOR iIndexInks:=1 TO MAX_LAST_INK DO
		gInks[iIndexInks].parameters.PrintheadsChiller.iIndex:=1; //Chiller is just for printheads, not inks.
	END_FOR

	//In case there were more than one curing led bar, two chiller are required
	IF iIndexWhiteCuringLedBar>1 OR iIndexColorCuringLedBar>1 OR iIndexPrimerCuringLedBar>1 THEN
		gMachine.Pt.Hw.iMaxNumChillers:=2;
	ELSE
		gMachine.Pt.Hw.iMaxNumChillers:=1;
	END_IF

	//Same type for all chillers
	FOR iChillerIndex:=1 TO gMachine.Pt.Hw.iMaxNumChillers DO
		gChiller[iChillerIndex].Parameters.xInstalled := TRUE;
		gChiller[iChillerIndex].Parameters.xEnable := TRUE;
		gChiller[iChillerIndex].Parameters.SystemType := CHILLERSYS_DIRECT;
	END_FOR

	//Camera
	gCamera.Parameters.xInstalled := TRUE; //Camera wont be considered as installed in water's machine type till hardware will be installed on those already manufactured machines
	gCamera.Parameters.iMappingBar := 10; //Located outside the block, after all printing and curing bars. So 9 index for mapping.

	// Powermeter
	gPowermeters[1].Parameters.xInstalled := TRUE;

	//Edge hold down
	gEdgeHoldDown.parameters.iAdjustmentSystemsNumber := 2; //1: Elevation, 2: Width fitting

	//Paired icla motors
	IF gMachine.Pt.ConfigNameID <> GC_CONFIG_SIMTEST_ID THEN
		gEdgeHoldDown.parameters.xInstalled := X20DIF371_180.ModuleOk;
		gPairedMotors[1].parameters.IndexIclaMaster :=3;
		gPairedMotors[1].parameters.IndexIclaGear :=5;
		gPairedMotors[2].parameters.IndexIclaMaster :=4;
		gPairedMotors[2].parameters.IndexIclaGear :=6;
	ELSE
		gEdgeHoldDown.parameters.xInstalled := TRUE;
		gPairedMotors[1].parameters.IndexIclaMaster :=4;
		gPairedMotors[1].parameters.IndexIclaGear :=5;
		gPairedMotors[2].parameters.IndexIclaMaster :=6;
		gPairedMotors[2].parameters.IndexIclaGear :=7;
	END_IF

	gPairedMotors[1].parameters.rMechPositionMin := 15;
	gPairedMotors[1].parameters.rMechPositionMax := 57;
	gPairedMotors[1].parameters.xPositionSensorInstalled := FALSE;
	gPairedMotors[1].parameters.JogSpeed:= 5;
	gPairedMotors[1].Motor[1].iDirection := -1;
	gPairedMotors[1].Motor[1].rHomePosition := (-1)*gPairedMotors[1].parameters.rMechPositionMin;
	gPairedMotors[1].Motor[2].iDirection := -1;
	gPairedMotors[1].Motor[2].rHomePosition := (-1)*gPairedMotors[1].parameters.rMechPositionMin;

	gPairedMotors[2].parameters.rMechPositionMin := 435;
	gPairedMotors[2].parameters.rMechPositionMax := 1430;
	gPairedMotors[2].parameters.xPositionSensorInstalled := TRUE;
	gPairedMotors[2].parameters.JogSpeed:= 3;
	gPairedMotors[2].Motor[1].iDirection := -1;
	gPairedMotors[2].Motor[1].rHomePosition := (-1)*gPairedMotors[2].parameters.rMechPositionMax;
	gPairedMotors[2].Motor[2].iDirection := 1;
	gPairedMotors[2].Motor[2].rHomePosition := gPairedMotors[2].parameters.rMechPositionMax;

	//Assgigning parameters to all adjustment systems
	FOR iIndexEhdSubsystems:=1 TO gEdgeHoldDown.parameters.iAdjustmentSystemsNumber DO
		gPairedMotors[iIndexEhdSubsystems].parameters.xInstalled := gEdgeHoldDown.status.xInstalled;
		gPairedMotors[iIndexEhdSubsystems].parameters.xEnabled := gEdgeHoldDown.status.xEnabled;

		gPairedMotors[iIndexEhdSubsystems].parameters.Acceleration:=5;
		gPairedMotors[iIndexEhdSubsystems].parameters.iNumIclaMotors := 2;

		gPairedMotors[iIndexEhdSubsystems].parameters.DriveUnit.ScrewPitch.PulsesPerTurn := 12;
		gPairedMotors[iIndexEhdSubsystems].parameters.DriveUnit.ScrewPitch.GearBox := 92;
	END_FOR

	gPairedMotors[1].parameters.Speed:=10;
	gPairedMotors[1].parameters.DriveUnit.ScrewPitch.Pitch := 4;
	gPairedMotors[1].parameters.DriveUnit.TransmissionType := TRANS_SCREW_PITCH;

	gPairedMotors[2].parameters.Speed:=300;
	gPairedMotors[2].parameters.DriveUnit.ScrewPitch.Pitch := 355;
	gPairedMotors[2].parameters.DriveUnit.TransmissionType := TRANS_LINEAL_PERIMETER;

	//LINE
	IF gMachine.Pt.ConfigNameID <> GC_CONFIG_SIMTEST_ID THEN
		gSarm.Parameters.xInstalled := Pdc_X20DIF371_050.ModuleOk;
	END_IF

	//External devices power managed from line's cabinet (PDC)
	gLine.Parameters.ExternalDevices[0].xIsEngine:=FALSE; 	//Printer
	gLine.Parameters.ExternalDevices[0].tiDelay := t#3s;
	gLine.Parameters.ExternalDevices[1].xIsEngine:=TRUE;	//Primer
	gLine.Parameters.ExternalDevices[1].tiDelay := t#60s;
	gLine.Parameters.ExternalDevices[2].xIsEngine:=FALSE;	//Feeder
	gLine.Parameters.ExternalDevices[2].tiDelay := t#3s;
	gLine.Parameters.ExternalDevices[3].xIsEngine:=TRUE;	//Dryer - IR1
	gLine.Parameters.ExternalDevices[3].tiDelay := t#3s;
	gLine.Parameters.ExternalDevices[4].xIsEngine:=TRUE;	//Dryer - IR2
	gLine.Parameters.ExternalDevices[4].tiDelay := t#3s;
	gLine.Parameters.ExternalDevices[5].xIsEngine:=FALSE; 	//Dryer controls
	gLine.Parameters.ExternalDevices[5].tiDelay := t#3s;
	gLine.Parameters.ExternalDevices[6].xIsEngine:=FALSE; 	//Stacker
	gLine.Parameters.ExternalDevices[6].tiDelay := t#3s;
	gLine.Parameters.ExternalDevices[7].xIsEngine:=FALSE; 	//UV
	gLine.Parameters.ExternalDevices[7].tiDelay := t#3s;
	gLine.Parameters.ExternalDevices[8].xIsEngine:=FALSE;	//Chiller
	gLine.Parameters.ExternalDevices[8].tiDelay := t#3s;
	gLine.Parameters.ExternalDevices[9].xIsEngine:=FALSE;	//Hoopers
	gLine.Parameters.ExternalDevices[9].tiDelay := t#3s;
	gLine.Parameters.ExternalDevices[10].xIsEngine:=TRUE;	//OPV
	gLine.Parameters.ExternalDevices[10].tiDelay := t#3s;
	gLine.Parameters.ExternalDevices[11].xIsEngine:=FALSE;	//Sarm
	gLine.Parameters.ExternalDevices[11].tiDelay := t#3s;

	// Assign total Devices
	gLine.Parameters.iNumExternalDevices := 11; //This is the trigger to start. Set the value once all others are properly assigned

	//SafetyController
	gSafetyController.Parameters.xInstalled := TRUE;

	/////////////////////////////////////////////////////
	/////   PLC CARDS	PLC CARDS	PLC CARDS	 ////////
	/////////////////////////////////////////////////////
	IF gPlcCards[0].Type <> CARD_UNDEFINED THEN
		RETURN;
	END_IF

	//Force "ModuleOk" in cards without it
	X20CPUData.ModuleOk := TRUE;

	//AsignCardsNozomi2;

END_ACTION
```

#### JamSensorsAssignation.st
```iecst
ACTION JamSensorsAssignation:

	IF NOT gMachine.parSw.xJamDetectEnable THEN
		RETURN;
	END_IF

	//Enable the jam sensor if a bar is installed in its position

	//Run the Jam devices
	FOR iIndexJamDevice := 1 TO gMachine.St.iJamDevices DO

		//Run the Jam sensors per device
		FOR iIndexJamSensor := 1 TO gMachine.Pt.CT.iNumSensorsPerJamDevice DO

			//Run the Inks to review if there is any of them with the same Mapping
			xIsBarInstalled := FALSE;
			CheckInkBarInJamPosition;
			gJamDetect[iIndexJamDevice].Parameters.xBarInstalled[iIndexJamSensor]:= xIsBarInstalled;

			//Run the curing led bars
			IF NOT xIsBarInstalled THEN
				CheckCuringBarInJamPosition;
				gJamDetect[iIndexJamDevice].Parameters.xBarInstalled[iIndexJamSensor]:= xIsBarInstalled;

				IF NOT xIsBarInstalled THEN
					CheckCameraInJamPosition;
					gJamDetect[iIndexJamDevice].Parameters.xBarInstalled[iIndexJamSensor]:= xIsBarInstalled;
				END_IF

			END_IF

		END_FOR

	END_FOR

END_ACTION

ACTION CheckInkBarInJamPosition:

	FOR iIndexInks :=1 TO MAX_LAST_INK DO

		//If there is a Match, mark it and return to avoid extra loops
		IF  gInks[iIndexInks].parSw.Config.iMappingBar = gJamDetect[iIndexJamDevice].Parameters.iMappingBarPos[iIndexJamSensor] AND
			gInks[iIndexInks].parSw.Config.iMappingBar > 0 THEN

			xIsBarInstalled := TRUE;

			gJamPerInk[iIndexInks].iJamDevice := iIndexJamDevice;
			gJamPerInk[iIndexInks].iJamSensor := iIndexJamSensor;

			RETURN;
		END_IF

	END_FOR

END_ACTION

ACTION CheckCuringBarInJamPosition:

	FOR iIndexCuringLedLamps :=1 TO MAX_LAST_CURING_LED DO

		//If there is a Match, mark it and return to avoid extra loops
		IF  gCuringLed[iIndexCuringLedLamps].Parameters.iMappingBar = gJamDetect[iIndexJamDevice].Parameters.iMappingBarPos[iIndexJamSensor] AND
			gCuringLed[iIndexCuringLedLamps].Parameters.xInstalled THEN

			xIsBarInstalled := TRUE;

			gJamPerCuringLed[iIndexCuringLedLamps].iJamDevice := iIndexJamDevice;
			gJamPerCuringLed[iIndexCuringLedLamps].iJamSensor := iIndexJamSensor;

			RETURN;
		END_IF

	END_FOR

END_ACTION

ACTION CheckCameraInJamPosition:

	IF  gCamera.Parameters.iMappingBar = gJamDetect[iIndexJamDevice].Parameters.iMappingBarPos[iIndexJamSensor] AND
		gCamera.Parameters.xInstalled THEN

		xIsBarInstalled := TRUE;

		gJamCamera.iJamDevice := iIndexJamDevice;
		gJamCamera.iJamSensor := iIndexJamSensor;

	END_IF

END_ACTION
```
